C07284=1039.411,-98.894,424.242,168.623,36.335,156.842
C07285=1039.404,-99.143,424.252,168.620,36.336,156.842
C07286=1039.399,-99.393,424.262,168.618,36.336,156.842
C07287=1039.392,-99.680,424.273,168.615,36.336,156.842
C07288=1039.384,-99.967,424.285,168.612,36.337,156.842
C07289=1039.378,-100.255,424.297,168.609,36.337,156.842
C07290=1039.371,-100.541,424.308,168.606,36.338,156.842
C07291=1039.364,-100.791,424.319,168.603,36.338,156.842
C07292=1039.358,-101.041,424.329,168.601,36.338,156.842
C07293=1039.352,-101.291,424.338,168.598,36.338,156.842
C07294=1039.346,-101.540,424.349,168.596,36.339,156.842
C07295=1039.340,-101.790,424.359,168.593,36.340,156.843
C07296=1039.334,-102.040,424.368,168.591,36.340,156.843
C07297=1039.328,-102.289,424.379,168.589,36.340,156.843
C07298=1039.322,-102.539,424.389,168.586,36.340,156.843
C07299=1039.316,-102.789,424.398,168.584,36.341,156.843
C07300=1039.310,-103.038,424.409,168.581,36.341,156.843
C07301=1039.303,-103.288,424.418,168.579,36.342,156.843
C07302=1039.298,-103.538,424.428,168.576,36.341,156.843
C07303=1039.291,-103.787,424.439,168.574,36.342,156.843
C07304=1039.285,-104.037,424.448,168.571,36.343,156.843
C07305=1039.279,-104.287,424.458,168.568,36.343,156.843
C07306=1039.274,-104.537,424.468,168.566,36.343,156.843
C07307=1039.267,-104.786,424.478,168.563,36.343,156.843
C07308=1039.261,-105.036,424.488,168.561,36.344,156.843
C07309=1039.255,-105.286,424.497,168.558,36.345,156.844
C07310=1039.249,-105.536,424.508,168.556,36.345,156.844
C07311=1039.243,-105.786,424.517,168.553,36.345,156.844
C07312=1039.237,-106.035,424.528,168.550,36.345,156.844
C07313=1039.231,-106.285,424.537,168.548,36.346,156.844
C07314=1039.224,-106.535,424.547,168.545,36.347,156.844
C07315=1039.219,-106.785,424.557,168.543,36.347,156.844
C07316=1039.213,-107.034,424.566,168.540,36.347,156.844
C07317=1039.207,-107.284,424.576,168.538,36.348,156.844
C07318=1039.200,-107.533,424.586,168.535,36.348,156.844
C07319=1039.194,-107.783,424.596,168.532,36.349,156.844
C07320=1039.188,-108.033,424.605,168.530,36.349,156.844
C07321=1039.182,-108.283,424.616,168.528,36.350,156.844
C07322=1039.176,-108.533,424.625,168.526,36.350,156.844
C07323=1039.170,-108.783,424.635,168.523,36.350,156.845
C07324=1039.164,-109.033,424.644,168.520,36.351,156.845
C07325=1039.158,-109.282,424.654,168.518,36.352,156.845
C07326=1039.152,-109.532,424.663,168.515,36.352,156.845
C07327=1039.146,-109.781,424.673,168.513,36.352,156.845
C07328=1039.140,-110.031,424.682,168.510,36.353,156.845
C07329=1039.134,-110.281,424.692,168.507,36.354,156.845
C07330=1039.127,-110.531,424.701,168.505,36.354,156.845
C07331=1039.121,-110.780,424.711,168.502,36.354,156.845
C07332=1039.115,-111.030,424.720,168.499,36.355,156.845
C07333=1039.109,-111.280,424.730,168.497,36.356,156.845
C07334=1039.103,-111.530,424.740,168.494,36.356,156.846
C07335=1039.097,-111.780,424.749,168.492,36.356,156.846
C07336=1039.090,-112.029,424.759,168.489,36.357,156.846
C07337=1039.086,-112.279,424.768,168.486,36.357,156.846
C07338=1039.079,-112.529,424.778,168.484,36.358,156.846
C07339=1039.073,-112.778,424.788,168.481,36.359,156.846
C07340=1039.067,-113.028,424.797,168.479,36.359,156.846
C07341=1039.061,-113.278,424.807,168.477,36.359,156.846
C07342=1039.055,-113.528,424.816,168.474,36.360,156.846
C07343=1039.049,-113.778,424.826,168.472,36.361,156.846
C07344=1039.043,-114.027,424.835,168.469,36.361,156.847
C07345=1039.037,-114.276,424.845,168.467,36.362,156.847
C07346=1039.031,-114.526,424.854,168.464,36.362,156.847
C07347=1039.025,-114.777,424.863,168.461,36.363,156.847
C07348=1039.019,-115.027,424.873,168.459,36.363,156.847
C07349=1039.012,-115.276,424.882,168.456,36.364,156.847
C07350=1039.007,-115.525,424.891,168.453,36.365,156.847
C07351=1038.999,-115.812,424.902,168.450,36.365,156.847
C07352=1038.993,-116.098,424.913,168.447,36.366,156.847
C07353=1038.985,-116.385,424.923,168.444,36.367,156.847
C07354=1038.979,-116.671,424.934,168.441,36.367,156.848
C07355=1038.972,-116.921,424.943,168.439,36.368,156.848
C07356=1038.967,-117.170,424.952,168.436,36.368,156.848
C07357=1038.961,-117.420,424.962,168.434,36.369,156.848
C07358=1038.954,-117.670,424.972,168.432,36.370,156.848
C07359=1038.949,-117.920,424.980,168.429,36.370,156.848
C07360=1038.942,-118.169,424.989,168.427,36.371,156.848
C07361=1038.936,-118.419,424.999,168.424,36.372,156.848
C07362=1038.930,-118.669,425.007,168.421,36.372,156.848
C07363=1038.924,-118.919,425.017,168.419,36.373,156.849
C07364=1038.918,-119.168,425.026,168.416,36.374,156.849
C07365=1038.912,-119.418,425.036,168.413,36.374,156.849
C07366=1038.906,-119.668,425.045,168.411,36.375,156.849
C07367=1038.900,-119.918,425.054,168.408,36.376,156.849
C07368=1038.894,-120.167,425.063,168.405,36.376,156.849
C07369=1038.888,-120.417,425.072,168.403,36.377,156.849
C07370=1038.882,-120.667,425.081,168.400,36.378,156.849
C07371=1038.876,-120.917,425.091,168.398,36.378,156.849
C07372=1038.870,-121.167,425.099,168.395,36.379,156.850
C07373=1038.864,-121.416,425.108,168.393,36.379,156.850
C07374=1038.858,-121.666,425.117,168.391,36.380,156.850
C07375=1038.852,-121.916,425.126,168.388,36.381,156.850
C07376=1038.846,-122.165,425.136,168.385,36.381,156.850
C07377=1038.840,-122.416,425.145,168.383,36.382,156.850
C07378=1038.834,-122.665,425.153,168.380,36.383,156.850
C07379=1038.828,-122.915,425.162,168.377,36.384,156.851
C07380=1038.822,-123.165,425.172,168.375,36.385,156.851
C07381=1038.816,-123.414,425.181,168.372,36.385,156.851
C07382=1038.810,-123.664,425.189,168.369,36.386,156.851
C07383=1038.803,-123.914,425.199,168.367,36.387,156.851
C07384=1038.798,-124.163,425.207,168.364,36.387,156.851
C07385=1038.792,-124.413,425.217,168.361,36.388,156.851
C07386=1038.785,-124.663,425.225,168.359,36.389,156.851
C07387=1038.780,-124.912,425.234,168.357,36.389,156.851
C07388=1038.774,-125.163,425.243,168.354,36.391,156.852
C07389=1038.767,-125.412,425.252,168.352,36.391,156.852
C07390=1038.762,-125.662,425.261,168.349,36.392,156.852
C07391=1038.756,-125.912,425.270,168.346,36.392,156.852
C07392=1038.750,-126.161,425.278,168.344,36.393,156.852
C07393=1038.744,-126.412,425.287,168.341,36.394,156.852
C07394=1038.738,-126.661,425.296,168.338,36.395,156.852
C07395=1038.732,-126.911,425.304,168.336,36.396,156.853
C07396=1038.725,-127.161,425.314,168.333,36.396,156.853
C07397=1038.720,-127.410,425.322,168.330,36.397,156.853
C07398=1038.714,-127.661,425.331,168.328,36.398,156.853
C07399=1038.708,-127.910,425.340,168.326,36.399,156.853
C07400=1038.703,-128.160,425.350,168.324,36.399,156.853
C07401=1038.698,-128.409,425.360,168.321,36.399,156.853
C07402=1038.695,-128.658,425.370,168.318,36.398,156.853
C07403=1038.692,-128.909,425.382,168.316,36.397,156.853
C07404=1038.690,-129.158,425.393,168.314,36.396,156.853
C07405=1038.689,-129.409,425.406,168.312,36.394,156.852
C07406=1038.689,-129.658,425.419,168.311,36.391,156.852
C07407=1038.690,-129.909,425.433,168.308,36.388,156.851
C07408=1038.690,-130.159,425.447,168.307,36.384,156.851
C07409=1038.692,-130.409,425.462,168.306,36.381,156.850
C07410=1038.695,-130.659,425.477,168.304,36.377,156.849
C07411=1038.698,-130.909,425.493,168.303,36.372,156.849
C07412=1038.703,-131.160,425.510,168.301,36.367,156.848
C07413=1038.707,-131.409,425.527,168.301,36.361,156.847
C07414=1038.713,-131.660,425.545,168.300,36.355,156.846
C07415=1038.372,-131.683,425.279,168.252,36.557,156.880
C07416=1038.366,-131.435,425.261,168.253,36.564,156.881
C07417=1038.360,-131.184,425.244,168.254,36.569,156.882
C07418=1038.356,-130.934,425.227,168.255,36.574,156.883
C07419=1038.353,-130.683,425.212,168.256,36.579,156.883
C07420=1038.350,-130.434,425.195,168.258,36.584,156.884
C07421=1038.348,-130.184,425.181,168.259,36.587,156.885
C07422=1038.347,-129.933,425.166,168.261,36.591,156.885
C07423=1038.346,-129.683,425.153,168.263,36.593,156.886
C07424=1038.347,-129.433,425.140,168.264,36.596,156.886
C07425=1038.349,-129.184,425.127,168.266,36.598,156.887
C07426=1038.350,-128.934,425.115,168.269,36.600,156.887
C07427=1038.352,-128.683,425.104,168.271,36.601,156.887
C07428=1038.357,-128.434,425.093,168.273,36.601,156.887
C07429=1038.361,-128.184,425.083,168.276,36.602,156.887
C07430=1038.365,-127.934,425.074,168.278,36.601,156.887
C07431=1038.371,-127.685,425.065,168.281,36.601,156.887
C07432=1038.377,-127.435,425.056,168.283,36.600,156.887
C07433=1038.383,-127.185,425.047,168.286,36.599,156.887
C07434=1038.389,-126.935,425.038,168.288,36.598,156.887
C07435=1038.395,-126.686,425.030,168.291,36.597,156.887
C07436=1038.401,-126.436,425.021,168.293,36.597,156.886
C07437=1038.407,-126.185,425.012,168.296,36.596,156.886
C07438=1038.413,-125.937,425.003,168.299,36.595,156.886
C07439=1038.419,-125.686,424.995,168.301,36.594,156.886
C07440=1038.425,-125.437,424.985,168.304,36.593,156.886
C07441=1038.431,-125.187,424.977,168.307,36.593,156.886
C07442=1038.437,-124.937,424.968,168.309,36.592,156.886
C07443=1038.443,-124.688,424.959,168.312,36.591,156.885
C07444=1038.450,-124.438,424.950,168.315,36.590,156.885
C07445=1038.455,-124.188,424.941,168.317,36.589,156.885
C07446=1038.461,-123.939,424.932,168.320,36.589,156.885
C07447=1038.467,-123.688,424.923,168.322,36.588,156.885
C07448=1038.474,-123.439,424.914,168.324,36.587,156.885
C07449=1038.479,-123.189,424.906,168.327,36.587,156.885
C07450=1038.485,-122.939,424.896,168.330,36.585,156.885
C07451=1038.491,-122.689,424.887,168.332,36.585,156.884
C07452=1038.497,-122.440,424.878,168.335,36.584,156.884
C07453=1038.504,-122.190,424.869,168.338,36.583,156.884
C07454=1038.509,-121.940,424.860,168.340,36.583,156.884
C07455=1038.515,-121.691,424.851,168.343,36.582,156.884
C07456=1038.521,-121.440,424.842,168.346,36.581,156.884
C07457=1038.527,-121.190,424.833,168.348,36.581,156.884
C07458=1038.533,-120.942,424.824,168.351,36.580,156.884
C07459=1038.539,-120.691,424.815,168.354,36.579,156.884
C07460=1038.545,-120.441,424.806,168.355,36.578,156.883
C07461=1038.551,-120.192,424.796,168.358,36.577,156.883
C07462=1038.557,-119.942,424.788,168.361,36.577,156.883
C07463=1038.563,-119.692,424.778,168.363,36.576,156.883
C07464=1038.570,-119.443,424.769,168.366,36.575,156.883
C07465=1038.575,-119.193,424.761,168.369,36.575,156.883
C07466=1038.581,-118.943,424.751,168.371,36.574,156.883
C07467=1038.587,-118.693,424.741,168.374,36.573,156.883
C07468=1038.593,-118.443,424.733,168.377,36.573,156.882
C07469=1038.599,-118.194,424.723,168.379,36.572,156.882
C07470=1038.605,-117.944,424.714,168.382,36.571,156.882
C07471=1038.612,-117.694,424.705,168.385,36.571,156.882
C07472=1038.618,-117.444,424.696,168.387,36.570,156.882
C07473=1038.623,-117.195,424.687,168.390,36.569,156.882
C07474=1038.630,-116.945,424.677,168.392,36.569,156.882
C07475=1038.636,-116.695,424.668,168.394,36.568,156.882
C07476=1038.642,-116.409,424.657,168.397,36.567,156.882
C07477=1038.650,-116.122,424.646,168.400,36.567,156.881
C07478=1038.657,-115.836,424.636,168.403,36.566,156.881
C07479=1038.663,-115.550,424.625,168.406,36.565,156.881
C07480=1038.670,-115.300,424.616,168.409,36.565,156.881
C07481=1038.676,-115.051,424.607,168.412,36.564,156.881
C07482=1038.682,-114.801,424.597,168.414,36.563,156.881
C07483=1038.688,-114.550,424.588,168.417,36.563,156.881
C07484=1038.694,-114.301,424.579,168.420,36.562,156.881
C07485=1038.700,-114.052,424.569,168.422,36.562,156.881
C07486=1038.706,-113.802,424.560,168.425,36.561,156.880
C07487=1038.712,-113.552,424.550,168.427,36.560,156.880
C07488=1038.718,-113.302,424.541,168.430,36.560,156.880
C07489=1038.724,-113.052,424.531,168.433,36.560,156.880
C07490=1038.730,-112.803,424.522,168.434,36.559,156.880
C07491=1038.736,-112.553,424.512,168.437,36.558,156.880
C07492=1038.742,-112.304,424.503,168.440,36.558,156.880
C07493=1038.748,-112.054,424.493,168.442,36.557,156.880
C07494=1038.753,-111.803,424.484,168.445,36.556,156.880
C07495=1038.760,-111.553,424.474,168.447,36.556,156.880
C07496=1038.766,-111.304,424.465,168.450,36.556,156.880
C07497=1038.772,-111.054,424.455,168.453,36.555,156.880
C07498=1038.778,-110.804,424.446,168.455,36.554,156.879
C07499=1038.784,-110.555,424.436,168.458,36.554,156.879
C07500=1038.790,-110.305,424.427,168.461,36.553,156.879
C07501=1038.796,-110.055,424.417,168.463,36.553,156.879
C07502=1038.802,-109.805,424.408,168.466,36.552,156.879
C07503=1038.809,-109.556,424.397,168.468,36.552,156.879
C07504=1038.815,-109.306,424.388,168.471,36.551,156.879
C07505=1038.821,-109.057,424.378,168.474,36.550,156.879
C07506=1038.827,-108.807,424.369,168.476,36.550,156.879
C07507=1038.833,-108.557,424.359,168.479,36.550,156.879
C07508=1038.840,-108.307,424.349,168.481,36.549,156.879
C07509=1038.845,-108.057,424.339,168.483,36.548,156.878
C07510=1038.851,-107.807,424.330,168.486,36.548,156.878
C07511=1038.857,-107.558,424.320,168.488,36.548,156.878
C07512=1038.864,-107.308,424.311,168.491,36.547,156.878
C07513=1038.870,-107.058,424.301,168.494,36.546,156.878
C07514=1038.876,-106.810,424.291,168.496,36.546,156.878
C07515=1038.882,-106.560,424.282,168.499,36.546,156.878
C07516=1038.887,-106.310,424.271,168.501,36.545,156.878
C07517=1038.893,-106.060,424.262,168.504,36.544,156.878
C07518=1038.900,-105.810,424.252,168.507,36.544,156.878
C07519=1038.906,-105.560,424.243,168.509,36.544,156.878
C07520=1038.911,-105.311,424.232,168.512,36.543,156.878
C07521=1038.918,-105.061,424.222,168.514,36.543,156.878
C07522=1038.924,-104.811,424.213,168.517,36.542,156.877
C07523=1038.930,-104.561,424.203,168.520,36.542,156.877
C07524=1038.936,-104.312,424.192,168.522,36.542,156.877
C07525=1038.942,-104.062,424.183,168.525,36.541,156.877
C07526=1038.948,-103.812,424.173,168.527,36.541,156.877
C07527=1038.954,-103.562,424.164,168.530,36.540,156.877
C07528=1038.960,-103.313,424.153,168.532,36.540,156.877
C07529=1038.966,-103.063,424.143,168.535,36.540,156.877
C07530=1038.972,-102.813,424.134,168.537,36.539,156.877
C07531=1038.979,-102.564,424.123,168.539,36.539,156.877
C07532=1038.985,-102.313,424.113,168.542,36.538,156.877
C07533=1038.991,-102.064,424.103,168.544,36.538,156.877
C07534=1038.997,-101.814,424.094,168.547,36.538,156.877
C07535=1039.003,-101.564,424.083,168.550,36.537,156.877
C07536=1039.009,-101.314,424.073,168.552,36.537,156.877
C07537=1039.016,-101.065,424.063,168.555,36.536,156.876
C07538=1039.022,-100.816,424.053,168.557,36.536,156.876
C07539=1039.027,-100.565,424.043,168.560,36.536,156.876
C07540=1039.035,-100.279,424.031,168.563,36.535,156.876
C07541=1039.042,-99.991,424.020,168.566,36.534,156.876
C07542=1039.049,-99.704,424.008,168.569,36.534,156.876
C07543=1039.055,-99.417,423.997,168.572,36.534,156.876
C07544=1039.062,-99.167,423.987,168.574,36.534,156.876
C07545=1039.068,-98.917,423.976,168.577,36.533,156.876
C07546=1039.074,-98.668,423.966,168.579,36.532,156.876
C07547=1039.081,-98.418,423.957,168.582,36.532,156.876
C07548=1039.086,-98.168,423.946,168.585,36.532,156.876
C07549=1039.092,-97.919,423.936,168.587,36.532,156.876
C07550=1039.099,-97.669,423.927,168.590,36.531,156.875
C07551=1039.105,-97.419,423.915,168.592,36.531,156.875
C07552=1039.111,-97.169,423.906,168.595,36.531,156.875
C07553=1039.117,-96.920,423.895,168.597,36.531,156.875
C07554=1039.123,-96.670,423.885,168.600,36.531,156.875
C07555=1039.129,-96.420,423.874,168.602,36.530,156.875
C07556=1039.135,-96.171,423.864,168.605,36.530,156.875
C07557=1039.141,-95.921,423.854,168.607,36.530,156.875
C07558=1039.146,-95.672,423.843,168.609,36.529,156.875
C07559=1039.153,-95.421,423.833,168.611,36.529,156.875
C07560=1039.159,-95.172,423.822,168.614,36.529,156.875
C07561=1039.165,-94.922,423.812,168.617,36.529,156.875
C07562=1039.171,-94.672,423.802,168.619,36.529,156.875
C07563=1039.177,-94.423,423.791,168.622,36.529,156.875
C07564=1039.183,-94.174,423.781,168.624,36.528,156.875
C07565=1039.189,-93.923,423.770,168.627,36.528,156.875
C07566=1039.196,-93.674,423.760,168.629,36.528,156.875
C07567=1039.201,-93.423,423.750,168.632,36.527,156.875
C07568=1039.207,-93.174,423.739,168.634,36.527,156.875
C07569=1039.213,-92.925,423.729,168.637,36.527,156.875
C07570=1039.219,-92.675,423.718,168.639,36.527,156.875
C07571=1039.226,-92.425,423.708,168.642,36.527,156.875
C07572=1039.231,-92.175,423.697,168.644,36.527,156.875
C07573=1039.238,-91.926,423.687,168.647,36.526,156.875
C07574=1039.243,-91.676,423.676,168.649,36.526,156.875
C07575=1039.250,-91.426,423.665,168.652,36.526,156.875
C07576=1039.256,-91.177,423.655,168.654,36.525,156.874
C07577=1039.262,-90.927,423.644,168.657,36.525,156.874
C07578=1039.268,-90.677,423.634,168.659,36.525,156.874
C07579=1039.274,-90.427,423.623,168.662,36.525,156.874
C07580=1039.280,-90.178,423.612,168.664,36.525,156.874
C07581=1039.287,-89.929,423.602,168.667,36.525,156.874
C07582=1039.292,-89.678,423.592,168.669,36.525,156.874
C07583=1039.299,-89.429,423.581,168.672,36.524,156.874
C07584=1039.305,-89.179,423.570,168.674,36.524,156.874
C07585=1039.311,-88.930,423.560,168.677,36.524,156.874
C07586=1039.318,-88.680,423.549,168.680,36.523,156.874
C07587=1039.323,-88.430,423.539,168.682,36.523,156.874
C07588=1039.329,-88.180,423.528,168.685,36.523,156.874
C07589=1039.335,-87.931,423.518,168.687,36.523,156.874
C07590=1039.342,-87.681,423.506,168.690,36.523,156.874
C07591=1039.348,-87.432,423.496,168.692,36.523,156.874
C07592=1039.354,-87.182,423.485,168.695,36.523,156.874
C07593=1039.360,-86.932,423.474,168.697,36.523,156.874
C07594=1039.366,-86.682,423.464,168.700,36.522,156.874
C07595=1039.372,-86.433,423.453,168.702,36.522,156.874
C07596=1039.379,-86.182,423.442,168.705,36.522,156.874
C07597=1039.385,-85.933,423.432,168.707,36.522,156.874
C07598=1039.391,-85.683,423.421,168.710,36.521,156.874
C07599=1039.397,-85.434,423.410,168.712,36.521,156.874
C07600=1039.404,-85.184,423.400,168.715,36.521,156.874
C07601=1039.410,-84.934,423.388,168.717,36.521,156.874
C07602=1039.416,-84.685,423.377,168.720,36.521,156.874
C07603=1039.422,-84.436,423.367,168.722,36.521,156.874
C07604=1039.429,-84.150,423.355,168.725,36.521,156.874
C07605=1039.437,-83.865,423.343,168.728,36.521,156.874
C07606=1039.444,-83.580,423.331,168.731,36.520,156.874
C07607=1039.450,-83.295,423.317,168.733,36.520,156.874
C07608=1039.457,-83.046,423.307,168.736,36.520,156.874
C07609=1039.463,-82.796,423.295,168.738,36.520,156.874
C07610=1039.469,-82.546,423.285,168.741,36.520,156.874
C07611=1039.476,-82.296,423.274,168.742,36.519,156.873
C07612=1039.482,-82.047,423.263,168.745,36.519,156.873
C07613=1039.488,-81.797,423.252,168.747,36.519,156.873
C07614=1039.495,-81.548,423.242,168.750,36.519,156.873
C07615=1039.501,-81.297,423.230,168.752,36.519,156.873
C07616=1039.507,-81.048,423.219,168.755,36.519,156.873
C07617=1039.513,-80.799,423.209,168.757,36.519,156.873
C07618=1039.519,-80.548,423.198,168.760,36.519,156.873
C07619=1039.525,-80.299,423.187,168.762,36.519,156.873
C07620=1039.532,-80.049,423.176,168.765,36.519,156.873
C07621=1039.538,-79.800,423.165,168.767,36.518,156.873
C07622=1039.545,-79.550,423.153,168.770,36.518,156.873
C07623=1039.550,-79.301,423.143,168.772,36.518,156.873
C07624=1039.557,-79.050,423.131,168.775,36.518,156.873
C07625=1039.563,-78.801,423.120,168.777,36.518,156.873
C07626=1039.569,-78.551,423.109,168.780,36.518,156.873
C07627=1039.575,-78.302,423.098,168.782,36.518,156.873
C07628=1039.581,-78.052,423.086,168.784,36.518,156.873
C07629=1039.587,-77.802,423.076,168.787,36.518,156.873
C07630=1039.593,-77.552,423.064,168.789,36.518,156.873
C07631=1039.600,-77.303,423.053,168.792,36.518,156.873
C07632=1039.606,-77.053,423.042,168.794,36.518,156.873
C07633=1039.612,-76.804,423.031,168.797,36.518,156.873
C07634=1039.619,-76.553,423.020,168.799,36.518,156.873
C07635=1039.625,-76.305,423.008,168.802,36.518,156.873
C07636=1039.631,-76.054,422.997,168.804,36.518,156.873
C07637=1039.637,-75.805,422.986,168.806,36.518,156.873
C07638=1039.643,-75.555,422.974,168.809,36.518,156.873
C07639=1039.649,-75.306,422.963,168.811,36.518,156.873
C07640=1039.655,-75.056,422.952,168.814,36.519,156.873
C07641=1039.662,-74.806,422.940,168.816,36.519,156.873
C07642=1039.668,-74.557,422.929,168.819,36.519,156.873
C07643=1039.674,-74.306,422.918,168.821,36.519,156.873
C07644=1039.680,-74.058,422.906,168.823,36.519,156.873
C07645=1039.686,-73.807,422.895,168.826,36.519,156.873
C07646=1039.692,-73.558,422.884,168.828,36.519,156.873
C07647=1039.699,-73.308,422.872,168.831,36.519,156.873
C07648=1039.704,-73.058,422.861,168.833,36.519,156.873
C07649=1039.711,-72.809,422.849,168.835,36.519,156.873
C07650=1039.717,-72.559,422.838,168.838,36.519,156.873
C07651=1039.723,-72.310,422.826,168.840,36.519,156.873
C07652=1039.729,-72.059,422.814,168.843,36.519,156.873
C07653=1039.735,-71.811,422.803,168.846,36.520,156.874
C07654=1039.741,-71.560,422.791,168.848,36.520,156.874
C07655=1039.747,-71.311,422.780,168.851,36.520,156.874
C07656=1039.753,-71.061,422.769,168.853,36.520,156.874
C07657=1039.759,-70.811,422.756,168.856,36.520,156.874
C07658=1039.765,-70.562,422.745,168.858,36.521,156.874
C07659=1039.772,-70.312,422.733,168.860,36.521,156.874
C07660=1039.777,-70.063,422.722,168.863,36.521,156.874
C07661=1039.783,-69.813,422.710,168.865,36.521,156.874
C07662=1039.790,-69.563,422.699,168.867,36.521,156.874
C07663=1039.796,-69.314,422.687,168.870,36.521,156.874
C07664=1039.802,-69.064,422.676,168.872,36.521,156.874
C07665=1039.807,-68.814,422.664,168.875,36.521,156.874
C07666=1039.814,-68.565,422.652,168.877,36.522,156.874
C07667=1039.820,-68.315,422.640,168.879,36.522,156.874
C07668=1039.827,-68.032,422.627,168.882,36.522,156.874
C07669=1039.834,-67.750,422.614,168.885,36.523,156.874
C07670=1039.841,-67.467,422.600,168.887,36.523,156.874
C07671=1039.848,-67.184,422.587,168.890,36.523,156.874
C07672=1039.855,-66.934,422.575,168.892,36.523,156.874
C07673=1039.860,-66.685,422.564,168.895,36.523,156.874
C07674=1039.866,-66.435,422.552,168.897,36.523,156.874
C07675=1039.873,-66.185,422.540,168.900,36.523,156.874
C07676=1039.878,-65.936,422.528,168.902,36.523,156.874
C07677=1039.885,-65.686,422.516,168.904,36.524,156.874
C07678=1039.891,-65.436,422.505,168.907,36.524,156.874
C07679=1039.897,-65.187,422.494,168.909,36.524,156.874
C07680=1039.903,-64.937,422.481,168.911,36.524,156.874
C07681=1039.910,-64.688,422.469,168.914,36.524,156.874
C07682=1039.916,-64.437,422.458,168.916,36.524,156.874
C07683=1039.921,-64.188,422.446,168.918,36.524,156.874
C07684=1039.928,-63.939,422.434,168.921,36.525,156.875
C07685=1039.935,-63.689,422.422,168.923,36.525,156.875
C07686=1039.941,-63.439,422.411,168.925,36.525,156.875
C07687=1039.946,-63.190,422.398,168.928,36.526,156.875
C07688=1039.953,-62.940,422.386,168.930,36.526,156.875
C07689=1039.960,-62.691,422.374,168.933,36.526,156.875
C07690=1039.965,-62.441,422.362,168.935,36.526,156.875
C07691=1039.971,-62.191,422.351,168.937,36.526,156.875
C07692=1039.978,-61.942,422.339,168.940,36.526,156.875
C07693=1039.984,-61.692,422.327,168.942,36.526,156.875
C07694=1039.990,-61.442,422.315,168.944,36.527,156.875
C07695=1039.997,-61.193,422.303,168.947,36.527,156.875
C07696=1040.003,-60.944,422.291,168.949,36.527,156.875
C07697=1040.009,-60.693,422.279,168.951,36.528,156.875
C07698=1040.015,-60.444,422.267,168.954,36.528,156.875
C07699=1040.022,-60.194,422.255,168.956,36.528,156.875
C07700=1040.028,-59.944,422.243,168.958,36.528,156.875
C07701=1040.035,-59.695,422.231,168.961,36.528,156.875
C07702=1040.041,-59.446,422.219,168.963,36.528,156.875
C07703=1040.046,-59.196,422.207,168.966,36.529,156.875
C07704=1040.053,-58.946,422.195,168.969,36.529,156.875
C07705=1040.059,-58.696,422.183,168.971,36.529,156.875
C07706=1040.065,-58.446,422.171,168.973,36.530,156.875
C07707=1040.072,-58.197,422.159,168.976,36.530,156.875
C07708=1040.079,-57.947,422.147,168.978,36.530,156.875
C07709=1040.084,-57.698,422.135,168.980,36.530,156.875
C07710=1040.091,-57.448,422.123,168.983,36.530,156.875
C07711=1040.097,-57.199,422.111,168.985,36.530,156.875
C07712=1040.103,-56.949,422.098,168.987,36.531,156.876
C07713=1040.110,-56.699,422.086,168.990,36.531,156.876
C07714=1040.116,-56.450,422.074,168.992,36.531,156.876
C07715=1040.122,-56.200,422.062,168.994,36.532,156.876
C07716=1040.129,-55.935,422.049,168.997,36.532,156.876
C07717=1040.136,-55.671,422.037,168.999,36.532,156.876
C07718=1040.143,-55.405,422.023,169.002,36.532,156.876
C07719=1040.150,-55.141,422.010,169.004,36.532,156.876
C07720=1040.156,-54.891,421.998,169.007,36.533,156.876
C07721=1040.162,-54.641,421.985,169.009,36.533,156.876
C07722=1040.169,-54.392,421.973,169.011,36.533,156.876
C07723=1040.175,-54.142,421.961,169.014,36.533,156.876
C07724=1040.181,-53.892,421.949,169.016,36.533,156.876
C07725=1040.188,-53.643,421.937,169.018,36.533,156.876
C07726=1040.194,-53.393,421.924,169.021,36.534,156.876
C07727=1040.201,-53.143,421.912,169.023,36.534,156.876
C07728=1040.207,-52.894,421.901,169.025,36.535,156.876
C07729=1040.213,-52.644,421.888,169.028,36.535,156.876
C07730=1040.220,-52.394,421.876,169.030,36.535,156.876
C07731=1040.226,-52.145,421.863,169.032,36.535,156.876
C07732=1040.233,-51.879,421.851,169.035,36.535,156.876
C07733=1040.239,-51.613,421.838,169.037,36.536,156.876
C07734=1040.247,-51.346,421.824,169.040,36.536,156.876
C07735=1040.253,-51.080,421.811,169.042,36.536,156.876
C07736=1040.260,-50.831,421.799,169.044,36.537,156.877
C07737=1040.266,-50.581,421.786,169.047,36.537,156.877
C07738=1040.272,-50.332,421.774,169.049,36.537,156.877
C07739=1040.278,-50.082,421.761,169.051,36.537,156.877
C07740=1040.284,-49.832,421.749,169.053,36.538,156.877
C07741=1040.291,-49.583,421.736,169.057,36.539,156.877
C07742=1040.297,-49.333,421.724,169.059,36.539,156.877
C07743=1040.303,-49.083,421.711,169.061,36.539,156.877
C07744=1040.309,-48.834,421.698,169.063,36.539,156.877
C07745=1040.316,-48.584,421.686,169.066,36.540,156.877
C07746=1040.322,-48.335,421.673,169.068,36.541,156.877
C07747=1040.328,-48.085,421.660,169.070,36.541,156.877
C07748=1040.334,-47.835,421.647,169.072,36.541,156.877
C07749=1040.341,-47.586,421.636,169.075,36.542,156.878
C07750=1040.347,-47.337,421.622,169.077,36.542,156.878
C07751=1040.353,-47.087,421.610,169.079,36.542,156.878
C07752=1040.359,-46.837,421.597,169.081,36.542,156.878
C07753=1040.366,-46.588,421.584,169.084,36.543,156.878
C07754=1040.372,-46.337,421.572,169.086,36.544,156.878
C07755=1040.378,-46.087,421.559,169.088,36.544,156.878
C07756=1040.384,-45.838,421.546,169.090,36.544,156.878
C07757=1040.391,-45.589,421.534,169.093,36.545,156.878
C07758=1040.397,-45.339,421.520,169.095,36.545,156.878
C07759=1040.403,-45.089,421.508,169.097,36.546,156.878
C07760=1040.409,-44.840,421.495,169.099,36.546,156.878
C07761=1040.416,-44.591,421.483,169.102,36.546,156.878
C07762=1040.422,-44.341,421.470,169.104,36.547,156.878
C07763=1040.428,-44.091,421.457,169.106,36.547,156.878
C07764=1040.434,-43.842,421.444,169.109,36.548,156.879
C07765=1040.441,-43.593,421.432,169.112,36.548,156.879
C07766=1040.447,-43.342,421.419,169.114,36.548,156.879
C07767=1040.454,-43.093,421.405,169.116,36.549,156.879
C07768=1040.459,-42.843,421.393,169.118,36.550,156.879
C07769=1040.466,-42.594,421.380,169.120,36.550,156.879
C07770=1040.472,-42.344,421.368,169.123,36.550,156.879
C07771=1040.479,-42.095,421.354,169.125,36.551,156.879
C07772=1040.484,-41.845,421.342,169.127,36.551,156.879
C07773=1040.491,-41.596,421.329,169.129,36.551,156.879
C07774=1040.497,-41.346,421.315,169.132,36.552,156.879
C07775=1040.504,-41.096,421.303,169.134,36.552,156.879
C07776=1040.510,-40.847,421.290,169.136,36.553,156.879
C07777=1040.516,-40.597,421.277,169.138,36.553,156.880
C07778=1040.522,-40.348,421.264,169.140,36.553,156.880
C07779=1040.529,-40.097,421.251,169.143,36.554,156.880
C07780=1040.536,-39.848,421.238,169.145,36.555,156.880
C07781=1040.542,-39.599,421.225,169.147,36.555,156.880
C07782=1040.548,-39.349,421.212,169.149,36.555,156.880
C07783=1040.554,-39.100,421.199,169.152,36.556,156.880
C07784=1040.561,-38.850,421.186,169.154,36.556,156.880
C07785=1040.567,-38.600,421.173,169.157,36.557,156.880
C07786=1040.573,-38.351,421.160,169.159,36.557,156.880
C07787=1040.579,-38.101,421.146,169.161,36.558,156.880
C07788=1040.585,-37.851,421.134,169.163,36.558,156.881
C07789=1040.592,-37.602,421.121,169.166,36.558,156.881
C07790=1040.598,-37.352,421.107,169.168,36.559,156.881
C07791=1040.604,-37.102,421.094,169.170,36.560,156.881
C07792=1040.610,-36.853,421.081,169.172,36.560,156.881
C07793=1040.617,-36.604,421.068,169.174,36.561,156.881
C07794=1040.623,-36.355,421.055,169.177,36.562,156.881
C07795=1040.629,-36.104,421.042,169.179,36.562,156.881
C07796=1040.636,-35.824,421.027,169.181,36.562,156.881
C07797=1040.643,-35.542,421.012,169.184,36.563,156.881
C07798=1040.651,-35.261,420.997,169.186,36.564,156.881
C07799=1040.657,-34.980,420.982,169.188,36.564,156.882
C07800=1040.664,-34.730,420.968,169.191,36.565,156.882
C07801=1040.670,-34.481,420.955,169.193,36.566,156.882
C07802=1040.676,-34.232,420.942,169.196,36.566,156.882
C07803=1040.683,-33.982,420.928,169.198,36.567,156.882
C07804=1040.689,-33.732,420.916,169.200,36.567,156.882
C07805=1040.695,-33.483,420.902,169.202,36.567,156.882
C07806=1040.701,-33.233,420.889,169.205,36.568,156.882
C07807=1040.708,-32.983,420.876,169.207,36.569,156.882
C07808=1040.714,-32.734,420.862,169.209,36.569,156.883
C07809=1040.720,-32.485,420.849,169.211,36.570,156.883
C07810=1040.727,-32.235,420.835,169.213,36.571,156.883
C07811=1040.733,-31.986,420.822,169.215,36.571,156.883
C07812=1040.740,-31.736,420.809,169.218,36.571,156.883
C07813=1040.745,-31.486,420.796,169.220,36.572,156.883
C07814=1040.752,-31.236,420.782,169.222,36.573,156.883
C07815=1040.758,-30.987,420.769,169.224,36.573,156.883
C07816=1040.764,-30.738,420.756,169.226,36.574,156.883
C07817=1040.771,-30.488,420.742,169.228,36.574,156.883
C07818=1040.777,-30.239,420.729,169.230,36.574,156.883
C07819=1040.783,-29.989,420.715,169.234,36.575,156.884
C07820=1040.790,-29.739,420.702,169.236,36.576,156.884
C07821=1040.796,-29.490,420.688,169.238,36.576,156.884
C07822=1040.803,-29.240,420.675,169.240,36.577,156.884
C07823=1040.809,-28.991,420.662,169.242,36.578,156.884
C07824=1040.815,-28.741,420.648,169.244,36.578,156.884
C07825=1040.822,-28.491,420.634,169.246,36.578,156.884
C07826=1040.828,-28.242,420.621,169.249,36.579,156.884
C07827=1040.834,-27.993,420.608,169.251,36.580,156.884
C07828=1040.841,-27.743,420.594,169.253,36.580,156.884
C07829=1040.847,-27.494,420.581,169.255,36.581,156.885
C07830=1040.854,-27.244,420.567,169.257,36.581,156.885
C07831=1040.860,-26.994,420.554,169.259,36.582,156.885
C07832=1040.866,-26.745,420.540,169.261,36.583,156.885
C07833=1040.873,-26.495,420.526,169.263,36.583,156.885
C07834=1040.879,-26.246,420.512,169.267,36.584,156.885
C07835=1040.884,-25.997,420.498,169.269,36.585,156.885
C07836=1040.891,-25.747,420.485,169.271,36.585,156.885
C07837=1040.897,-25.497,420.471,169.273,36.586,156.886
C07838=1040.904,-25.247,420.457,169.275,36.587,156.886
C07839=1040.910,-24.998,420.444,169.277,36.587,156.886
C07840=1040.916,-24.749,420.429,169.279,36.588,156.886
C07841=1040.922,-24.499,420.416,169.281,36.589,156.886
C07842=1040.929,-24.250,420.402,169.283,36.589,156.886
C07843=1040.935,-23.999,420.388,169.285,36.590,156.886
C07844=1040.941,-23.750,420.375,169.288,36.590,156.886
C07845=1040.947,-23.501,420.361,169.290,36.591,156.886
C07846=1040.953,-23.251,420.347,169.292,36.592,156.887
C07847=1040.960,-23.002,420.333,169.294,36.592,156.887
C07848=1040.966,-22.752,420.320,169.297,36.593,156.887
C07849=1040.972,-22.503,420.305,169.299,36.594,156.887
C07850=1040.979,-22.253,420.292,169.301,36.594,156.887
C07851=1040.985,-22.003,420.278,169.303,36.595,156.887
C07852=1040.991,-21.753,420.264,169.305,36.596,156.887
C07853=1040.998,-21.505,420.250,169.307,36.596,156.887
C07854=1041.004,-21.255,420.236,169.309,36.597,156.888
C07855=1041.010,-21.005,420.223,169.311,36.597,156.888
C07856=1041.017,-20.756,420.208,169.314,36.598,156.888
C07857=1041.023,-20.506,420.194,169.316,36.599,156.888
C07858=1041.030,-20.256,420.181,169.318,36.599,156.888
C07859=1041.035,-20.007,420.167,169.320,36.600,156.888
C07860=1041.043,-19.725,420.151,169.322,36.601,156.888
C07861=1041.050,-19.444,420.135,169.324,36.601,156.888
C07862=1041.057,-19.161,420.120,169.328,36.603,156.889
C07863=1041.064,-18.880,420.104,169.330,36.603,156.889
C07864=1041.070,-18.630,420.090,169.332,36.604,156.889
C07865=1041.077,-18.381,420.075,169.334,36.604,156.889
C07866=1041.083,-18.131,420.062,169.336,36.605,156.889
C07867=1041.089,-17.881,420.048,169.338,36.606,156.889
C07868=1041.096,-17.632,420.034,169.340,36.606,156.889
C07869=1041.102,-17.383,420.020,169.343,36.607,156.889
C07870=1041.109,-17.133,420.005,169.345,36.608,156.890
C07871=1041.115,-16.884,419.992,169.347,36.608,156.890
C07872=1041.121,-16.634,419.977,169.349,36.609,156.890
C07873=1041.128,-16.385,419.964,169.351,36.610,156.890
C07874=1041.134,-16.135,419.950,169.353,36.610,156.890
C07875=1041.140,-15.886,419.936,169.356,36.611,156.890
C07876=1041.147,-15.636,419.922,169.358,36.611,156.890
C07877=1041.153,-15.386,419.907,169.360,36.612,156.890
C07878=1041.160,-15.137,419.894,169.362,36.613,156.890
C07879=1041.166,-14.887,419.879,169.364,36.614,156.891
C07880=1041.172,-14.638,419.865,169.366,36.615,156.891
C07881=1041.179,-14.388,419.851,169.368,36.615,156.891
C07882=1041.184,-14.139,419.837,169.370,36.616,156.891
C07883=1041.191,-13.889,419.822,169.372,36.617,156.891
C07884=1041.198,-13.640,419.807,169.374,36.617,156.891
C07885=1041.203,-13.390,419.794,169.376,36.618,156.891
C07886=1041.210,-13.140,419.779,169.378,36.619,156.892
C07887=1041.216,-12.891,419.765,169.381,36.620,156.892
C07888=1041.222,-12.642,419.750,169.383,36.620,156.892
C07889=1041.228,-12.392,419.735,169.385,36.621,156.892
C07890=1041.235,-12.143,419.722,169.387,36.622,156.892
C07891=1041.241,-11.893,419.707,169.389,36.623,156.892
C07892=1041.247,-11.643,419.693,169.391,36.623,156.892
C07893=1041.254,-11.394,419.679,169.393,36.624,156.893
C07894=1041.260,-11.144,419.664,169.395,36.625,156.893
C07895=1041.266,-10.895,419.650,169.397,36.625,156.893
C07896=1041.273,-10.645,419.636,169.399,36.627,156.893
C07897=1041.279,-10.396,419.621,169.401,36.627,156.893
C07898=1041.285,-10.146,419.607,169.403,36.628,156.893
C07899=1041.292,-9.897,419.593,169.406,36.629,156.893
C07900=1041.298,-9.647,419.578,169.408,36.629,156.893
C07901=1041.304,-9.398,419.563,169.410,36.630,156.894
C07902=1041.311,-9.148,419.550,169.412,36.631,156.894
C07903=1041.317,-8.899,419.535,169.414,36.632,156.894
C07904=1041.323,-8.650,419.520,169.416,36.632,156.894
C07905=1041.330,-8.400,419.506,169.418,36.633,156.894
C07906=1041.336,-8.150,419.491,169.420,36.634,156.894
C07907=1041.342,-7.901,419.477,169.422,36.635,156.895
C07908=1041.348,-7.651,419.462,169.424,36.636,156.895
C07909=1041.355,-7.402,419.448,169.426,36.636,156.895
C07910=1041.361,-7.153,419.434,169.428,36.637,156.895
C07911=1041.367,-6.903,419.419,169.431,36.637,156.895
C07912=1041.374,-6.654,419.404,169.433,36.639,156.895
C07913=1041.381,-6.404,419.389,169.435,36.639,156.895
C07914=1041.386,-6.154,419.376,169.437,36.640,156.895
C07915=1041.393,-5.905,419.361,169.439,36.641,156.896
C07916=1041.400,-5.655,419.346,169.441,36.641,156.896
C07917=1041.405,-5.406,419.332,169.443,36.642,156.896
C07918=1041.412,-5.157,419.317,169.445,36.643,156.896
C07919=1041.419,-4.907,419.302,169.447,36.644,156.896
C07920=1041.425,-4.657,419.288,169.449,36.644,156.896
C07921=1041.431,-4.407,419.273,169.451,36.645,156.896
C07922=1041.437,-4.158,419.259,169.453,36.646,156.897
C07923=1041.444,-3.909,419.244,169.456,36.647,156.897
C07924=1041.451,-3.626,419.228,169.459,36.648,156.897
C07925=1041.459,-3.343,419.211,169.461,36.648,156.897
C07926=1041.466,-3.058,419.194,169.463,36.649,156.897
C07927=1041.473,-2.775,419.177,169.465,36.651,156.897
C07928=1041.479,-2.526,419.163,169.467,36.651,156.898
C07929=1041.485,-2.276,419.148,169.469,36.652,156.898
C07930=1041.491,-2.027,419.133,169.471,36.653,156.898
C07931=1041.498,-1.777,419.118,169.473,36.654,156.898
C07932=1041.503,-1.528,419.103,169.476,36.655,156.898
C07933=1041.510,-1.278,419.088,169.478,36.656,156.898
C07934=1041.516,-1.029,419.073,169.480,36.656,156.899
C07935=1041.523,-0.779,419.058,169.482,36.658,156.899
C07936=1041.529,-0.531,419.043,169.484,36.658,156.899
C07937=1041.535,-0.281,419.028,169.486,36.659,156.899
C07938=1041.541,-0.031,419.013,169.488,36.660,156.899
C07939=1041.547,0.219,418.998,169.489,36.661,156.899
C07940=1041.553,0.468,418.983,169.491,36.662,156.899
C07941=1041.559,0.717,418.968,169.493,36.663,156.900
C07942=1041.566,0.967,418.953,169.496,36.663,156.900
C07943=1041.572,1.217,418.938,169.498,36.664,156.900
C07944=1041.578,1.466,418.923,169.500,36.665,156.900
C07945=1041.585,1.716,418.908,169.502,36.666,156.900
C07946=1041.591,1.965,418.894,169.504,36.667,156.901
C07947=1041.597,2.214,418.879,169.506,36.668,156.901
C07948=1041.604,2.464,418.863,169.508,36.668,156.901
C07949=1041.610,2.713,418.848,169.510,36.670,156.901
C07950=1041.616,2.963,418.833,169.512,36.670,156.901
C07951=1041.622,3.212,418.819,169.514,36.671,156.901
C07952=1041.629,3.461,418.804,169.517,36.672,156.902
C07953=1041.635,3.711,418.789,169.518,36.673,156.902
C07954=1041.642,3.960,418.773,169.520,36.674,156.902
C07955=1041.647,4.210,418.758,169.522,36.675,156.902
C07956=1041.654,4.460,418.743,169.524,36.675,156.902
C07957=1041.660,4.709,418.728,169.526,36.677,156.902
C07958=1041.666,4.959,418.713,169.528,36.677,156.902
C07959=1041.673,5.207,418.697,169.530,36.678,156.903
C07960=1041.679,5.457,418.683,169.532,36.679,156.903
C07961=1041.685,5.707,418.668,169.534,36.680,156.903
C07962=1041.692,5.956,418.653,169.537,36.680,156.903
C07963=1041.698,6.205,418.637,169.539,36.682,156.903
C07964=1041.705,6.455,418.622,169.541,36.682,156.903
C07965=1041.711,6.705,418.607,169.542,36.683,156.904
C07966=1041.718,6.954,418.592,169.544,36.684,156.904
C07967=1041.723,7.204,418.576,169.546,36.685,156.904
C07968=1041.730,7.453,418.561,169.548,36.686,156.904
C07969=1041.736,7.703,418.546,169.550,36.687,156.904
C07970=1041.742,7.951,418.531,169.552,36.687,156.904
C07971=1041.749,8.201,418.516,169.554,36.689,156.905
C07972=1041.755,8.451,418.501,169.557,36.689,156.905
C07973=1041.761,8.700,418.486,169.559,36.690,156.905
C07974=1041.768,8.949,418.470,169.561,36.691,156.905
C07975=1041.775,9.199,418.455,169.563,36.692,156.905
C07976=1041.780,9.449,418.440,169.564,36.692,156.905
C07977=1041.787,9.698,418.424,169.566,36.694,156.906
C07978=1041.793,9.948,418.409,169.568,36.694,156.906
C07979=1041.800,10.197,418.393,169.570,36.695,156.906
C07980=1041.806,10.446,418.378,169.572,36.696,156.906
C07981=1041.813,10.696,418.364,169.574,36.697,156.906
C07982=1041.819,10.945,418.348,169.576,36.698,156.906
C07983=1041.826,11.195,418.333,169.579,36.699,156.906
C07984=1041.833,11.444,418.317,169.581,36.699,156.907
C07985=1041.838,11.694,418.302,169.583,36.700,156.907
C07986=1041.845,11.943,418.287,169.585,36.701,156.907
C07987=1041.851,12.192,418.271,169.586,36.702,156.907
C07988=1041.859,12.478,418.253,169.589,36.703,156.907
C07989=1041.866,12.764,418.236,169.591,36.704,156.907
C07990=1041.874,13.049,418.219,169.593,36.705,156.908
C07991=1041.881,13.334,418.201,169.595,36.706,156.908
C07992=1041.887,13.584,418.186,169.598,36.707,156.908
C07993=1041.893,13.833,418.170,169.600,36.708,156.908
C07994=1041.900,14.083,418.155,169.602,36.708,156.908
C07995=1041.906,14.332,418.139,169.604,36.709,156.908
C07996=1041.913,14.581,418.124,169.606,36.710,156.909
C07997=1041.919,14.831,418.108,169.607,36.711,156.909
C07998=1041.925,15.080,418.092,169.609,36.712,156.909
C07999=1041.931,15.330,418.077,169.611,36.713,156.909
C08000=1041.938,15.579,418.061,169.613,36.714,156.909
C08001=1041.944,15.828,418.046,169.616,36.715,156.910
C08002=1041.950,16.078,418.030,169.618,36.716,156.910
C08003=1041.957,16.327,418.014,169.620,36.717,156.910
C08004=1041.962,16.577,417.999,169.621,36.718,156.910
C08005=1041.969,16.826,417.983,169.623,36.719,156.910
C08006=1041.976,17.076,417.968,169.625,36.720,156.910
C08007=1041.982,17.325,417.952,169.627,36.721,156.911
C08008=1041.989,17.575,417.936,169.629,36.721,156.911
C08009=1041.994,17.824,417.920,169.631,36.723,156.911
C08010=1042.001,18.074,417.905,169.634,36.723,156.911
C08011=1042.008,18.323,417.889,169.635,36.725,156.911
C08012=1042.013,18.573,417.874,169.637,36.725,156.911
C08013=1042.020,18.822,417.858,169.639,36.726,156.912
C08014=1042.026,19.071,417.842,169.641,36.727,156.912
C08015=1042.032,19.321,417.827,169.643,36.728,156.912
C08016=1042.039,19.570,417.811,169.645,36.729,156.912
C08017=1042.045,19.819,417.795,169.647,36.730,156.912
C08018=1042.052,20.069,417.779,169.648,36.731,156.913
C08019=1042.058,20.319,417.763,169.651,36.732,156.913
C08020=1042.065,20.568,417.748,169.653,36.733,156.913
C08021=1042.071,20.817,417.731,169.655,36.734,156.913
C08022=1042.077,21.066,417.716,169.657,36.735,156.913
C08023=1042.083,21.316,417.700,169.659,36.736,156.913
C08024=1042.090,21.565,417.684,169.660,36.737,156.914
C08025=1042.096,21.814,417.668,169.662,36.738,156.914
C08026=1042.102,22.064,417.652,169.664,36.738,156.914
C08027=1042.109,22.314,417.636,169.666,36.740,156.914
C08028=1042.115,22.563,417.620,169.669,36.740,156.914
C08029=1042.121,22.813,417.605,169.671,36.742,156.915
C08030=1042.127,23.062,417.588,169.672,36.742,156.915
C08031=1042.134,23.311,417.573,169.674,36.743,156.915
C08032=1042.140,23.560,417.556,169.676,36.744,156.915
C08033=1042.147,23.809,417.541,169.678,36.745,156.915
C08034=1042.153,24.060,417.525,169.680,36.746,156.915
C08035=1042.159,24.309,417.509,169.681,36.747,156.916
C08036=1042.165,24.558,417.493,169.684,36.748,156.916
C08037=1042.171,24.808,417.477,169.686,36.749,156.916
C08038=1042.178,25.057,417.461,169.688,36.750,156.916
C08039=1042.185,25.307,417.444,169.690,36.751,156.916
C08040=1042.191,25.556,417.429,169.692,36.752,156.917
C08041=1042.197,25.805,417.413,169.693,36.753,156.917
C08042=1042.204,26.054,417.397,169.695,36.754,156.917
C08043=1042.210,26.304,417.381,169.697,36.755,156.917
C08044=1042.216,26.554,417.364,169.699,36.756,156.917
C08045=1042.223,26.803,417.349,169.702,36.757,156.917
C08046=1042.229,27.053,417.333,169.704,36.758,156.918
C08047=1042.235,27.302,417.317,169.705,36.759,156.918
C08048=1042.241,27.551,417.301,169.707,36.760,156.918
C08049=1042.248,27.801,417.284,169.709,36.760,156.918
C08050=1042.255,28.050,417.269,169.711,36.762,156.918
C08051=1042.261,28.299,417.252,169.713,36.763,156.919
C08052=1042.268,28.586,417.234,169.715,36.764,156.919
C08053=1042.275,28.872,417.214,169.718,36.765,156.919
C08054=1042.282,29.160,417.196,169.720,36.766,156.919
C08055=1042.290,29.446,417.178,169.722,36.767,156.919
C08056=1042.296,29.695,417.161,169.724,36.769,156.920
C08057=1042.302,29.945,417.145,169.725,36.769,156.920
C08058=1042.308,30.194,417.129,169.727,36.770,156.920
C08059=1042.315,30.444,417.113,169.729,36.772,156.920
C08060=1042.321,30.693,417.096,169.731,36.772,156.920
C08061=1042.327,30.942,417.079,169.734,36.774,156.921
C08062=1042.333,31.191,417.063,169.735,36.774,156.921
C08063=1042.340,31.441,417.047,169.737,36.775,156.921
C08064=1042.346,31.690,417.031,169.739,36.777,156.921
C08065=1042.352,31.940,417.015,169.741,36.777,156.921
C08066=1042.358,32.189,416.998,169.743,36.779,156.922
C08067=1042.365,32.438,416.981,169.744,36.780,156.922
C08068=1042.372,32.688,416.965,169.746,36.780,156.922
C08069=1042.378,32.937,416.949,169.749,36.782,156.922
C08070=1042.384,33.187,416.933,169.751,36.782,156.922
C08071=1042.390,33.436,416.916,169.753,36.784,156.923
C08072=1042.396,33.686,416.900,169.754,36.785,156.923
C08073=1042.402,33.934,416.883,169.756,36.785,156.923
C08074=1042.410,34.184,416.867,169.758,36.787,156.923
C08075=1042.416,34.433,416.851,169.760,36.787,156.923
C08076=1042.422,34.683,416.835,169.762,36.789,156.924
C08077=1042.428,34.933,416.818,169.764,36.790,156.924
C08078=1042.434,35.182,416.801,169.766,36.790,156.924
C08079=1042.441,35.431,416.785,169.768,36.792,156.924
C08080=1042.448,35.681,416.769,169.770,36.792,156.924
C08081=1042.454,35.930,416.752,169.771,36.794,156.924
C08082=1042.460,36.179,416.735,169.773,36.795,156.925
C08083=1042.466,36.429,416.719,169.775,36.795,156.925
C08084=1042.472,36.678,416.703,169.777,36.797,156.925
C08085=1042.479,36.927,416.686,169.779,36.797,156.925
C08086=1042.486,37.177,416.670,169.781,36.799,156.925
C08087=1042.492,37.426,416.653,169.783,36.800,156.926
C08088=1042.498,37.675,416.637,169.785,36.800,156.926
C08089=1042.505,37.925,416.620,169.787,36.802,156.926
C08090=1042.511,38.174,416.603,169.788,36.803,156.926
C08091=1042.517,38.423,416.586,169.790,36.804,156.926
C08092=1042.523,38.673,416.570,169.792,36.805,156.927
C08093=1042.529,38.922,416.554,169.795,36.806,156.927
C08094=1042.536,39.172,416.536,169.797,36.807,156.927
C08095=1042.542,39.421,416.520,169.798,36.808,156.927
C08096=1042.548,39.670,416.504,169.800,36.809,156.927
C08097=1042.554,39.920,416.486,169.802,36.810,156.928
C08098=1042.560,40.169,416.470,169.804,36.811,156.928
C08099=1042.566,40.418,416.453,169.805,36.812,156.928
C08100=1042.573,40.668,416.436,169.807,36.814,156.928
C08101=1042.579,40.917,416.419,169.810,36.814,156.928
C08102=1042.586,41.167,416.402,169.812,36.815,156.929
C08103=1042.592,41.416,416.385,169.813,36.817,156.929
C08104=1042.598,41.665,416.369,169.815,36.818,156.929
C08105=1042.605,41.915,416.353,169.817,36.819,156.929
C08106=1042.611,42.164,416.336,169.819,36.820,156.930
C08107=1042.617,42.414,416.319,169.820,36.821,156.930
C08108=1042.624,42.663,416.302,169.822,36.822,156.930
C08109=1042.630,42.912,416.286,169.825,36.823,156.930
C08110=1042.636,43.161,416.268,169.827,36.824,156.930
C08111=1042.643,43.410,416.251,169.828,36.825,156.930
C08112=1042.649,43.660,416.234,169.830,36.826,156.931
C08113=1042.655,43.909,416.217,169.832,36.827,156.931
C08114=1042.661,44.159,416.201,169.834,36.829,156.931
C08115=1042.667,44.408,416.183,169.835,36.830,156.931
C08116=1042.674,44.695,416.164,169.838,36.831,156.932
C08117=1042.681,44.980,416.144,169.840,36.832,156.932
C08118=1042.688,45.268,416.125,169.842,36.834,156.932
C08119=1042.695,45.554,416.106,169.844,36.835,156.932
C08120=1042.701,45.804,416.088,169.846,36.836,156.933
C08121=1042.708,46.053,416.071,169.848,36.837,156.933
C08122=1042.713,46.302,416.054,169.850,36.838,156.933
C08123=1042.720,46.552,416.037,169.852,36.839,156.933
C08124=1042.726,46.801,416.019,169.854,36.840,156.933
C08125=1042.732,47.051,416.003,169.856,36.842,156.934
C08126=1042.739,47.299,415.986,169.857,36.843,156.934
C08127=1042.745,47.549,415.968,169.859,36.844,156.934
C08128=1042.751,47.798,415.952,169.861,36.845,156.934
C08129=1042.758,48.048,415.934,169.864,36.846,156.935
C08130=1042.763,48.297,415.917,169.865,36.847,156.935
C08131=1042.770,48.546,415.899,169.867,36.849,156.935
C08132=1042.776,48.796,415.883,169.869,36.850,156.935
C08133=1042.781,49.045,415.866,169.870,36.850,156.935
C08134=1042.788,49.294,415.848,169.872,36.852,156.936
C08135=1042.794,49.544,415.832,169.874,36.853,156.936
C08136=1042.800,49.793,415.814,169.877,36.854,156.936
C08137=1042.807,50.042,415.797,169.878,36.855,156.936
C08138=1042.813,50.291,415.780,169.880,36.856,156.937
C08139=1042.819,50.540,415.762,169.882,36.857,156.937
C08140=1042.826,50.791,415.746,169.884,36.859,156.937
C08141=1042.831,51.040,415.728,169.885,36.860,156.937
C08142=1042.838,51.289,415.711,169.887,36.860,156.937
C08143=1042.844,51.538,415.694,169.889,36.862,156.938
C08144=1042.850,51.787,415.676,169.891,36.863,156.938
C08145=1042.857,52.038,415.659,169.893,36.864,156.938
C08146=1042.863,52.286,415.642,169.895,36.865,156.938
C08147=1042.869,52.536,415.624,169.897,36.866,156.938
C08148=1042.875,52.785,415.607,169.898,36.867,156.939
C08149=1042.882,53.034,415.590,169.900,36.869,156.939
C08150=1042.888,53.283,415.572,169.902,36.870,156.939
C08151=1042.894,53.533,415.556,169.905,36.870,156.939
C08152=1042.900,53.782,415.538,169.906,36.872,156.940
C08153=1042.907,54.032,415.521,169.908,36.873,156.940
C08154=1042.914,54.281,415.504,169.910,36.874,156.940
C08155=1042.919,54.530,415.486,169.911,36.875,156.940
C08156=1042.926,54.780,415.469,169.913,36.876,156.940
C08157=1042.932,55.028,415.452,169.915,36.877,156.941
C08158=1042.938,55.278,415.434,169.918,36.878,156.941
C08159=1042.945,55.527,415.416,169.919,36.879,156.941
C08160=1042.951,55.777,415.399,169.921,36.880,156.941
C08161=1042.958,56.026,415.381,169.923,36.882,156.941
C08162=1042.964,56.275,415.365,169.925,36.883,156.942
C08163=1042.970,56.525,415.347,169.926,36.883,156.942
C08164=1042.977,56.774,415.330,169.928,36.885,156.942
C08165=1042.983,57.023,415.313,169.931,36.886,156.942
C08166=1042.989,57.273,415.295,169.933,36.887,156.943
C08167=1042.996,57.522,415.278,169.934,36.888,156.943
C08168=1043.001,57.771,415.260,169.936,36.889,156.943
C08169=1043.008,58.021,415.243,169.938,36.890,156.943
C08170=1043.014,58.270,415.226,169.939,36.892,156.943
C08171=1043.021,58.519,415.208,169.941,36.892,156.944
C08172=1043.027,58.769,415.191,169.943,36.893,156.944
C08173=1043.033,59.018,415.173,169.946,36.895,156.944
C08174=1043.040,59.267,415.156,169.947,36.896,156.944
C08175=1043.047,59.517,415.138,169.949,36.897,156.944
C08176=1043.052,59.765,415.120,169.951,36.898,156.945
C08177=1043.059,60.014,415.103,169.953,36.899,156.945
C08178=1043.065,60.264,415.085,169.954,36.900,156.945
C08179=1043.072,60.514,415.067,169.956,36.901,156.945
C08180=1043.079,60.800,415.047,169.959,36.902,156.945
C08181=1043.087,61.086,415.027,169.961,36.903,156.946
C08182=1043.094,61.372,415.007,169.963,36.905,156.946
C08183=1043.101,61.659,414.987,169.965,36.906,156.946
C08184=1043.108,61.908,414.970,169.967,36.907,156.946
C08185=1043.114,62.157,414.952,169.969,36.908,156.947
C08186=1043.121,62.407,414.935,169.970,36.909,156.947
C08187=1043.127,62.656,414.917,169.973,36.910,156.947
C08188=1043.133,62.905,414.899,169.975,36.911,156.947
C08189=1043.140,63.154,414.882,169.977,36.912,156.947
C08190=1043.146,63.404,414.864,169.978,36.913,156.948
C08191=1043.153,63.653,414.846,169.980,36.914,156.948
C08192=1043.159,63.902,414.829,169.982,36.915,156.948
C08193=1043.166,64.152,414.812,169.984,36.916,156.948
C08194=1043.172,64.401,414.793,169.986,36.918,156.949
C08195=1043.178,64.651,414.775,169.988,36.919,156.949
C08196=1043.184,64.899,414.758,169.990,36.920,156.949
C08197=1043.190,65.149,414.740,169.991,36.921,156.949
C08198=1043.197,65.398,414.721,169.993,36.922,156.949
C08199=1043.202,65.647,414.704,169.995,36.923,156.950
C08200=1043.209,65.897,414.686,169.996,36.924,156.950
C08201=1043.216,66.146,414.668,169.999,36.926,156.950
C08202=1043.222,66.395,414.650,170.001,36.927,156.950
C08203=1043.228,66.644,414.633,170.003,36.928,156.951
C08204=1043.234,66.894,414.615,170.004,36.929,156.951
C08205=1043.241,67.143,414.596,170.006,36.930,156.951
C08206=1043.247,67.392,414.579,170.008,36.931,156.951
C08207=1043.253,67.641,414.561,170.010,36.932,156.951
C08208=1043.259,67.891,414.543,170.012,36.934,156.952
C08209=1043.265,68.140,414.525,170.014,36.935,156.952
C08210=1043.273,68.389,414.507,170.016,36.936,156.952
C08211=1043.278,68.638,414.489,170.017,36.937,156.952
C08212=1043.284,68.888,414.471,170.019,36.938,156.953
C08213=1043.291,69.137,414.453,170.021,36.939,156.953
C08214=1043.298,69.387,414.435,170.023,36.941,156.953
C08215=1043.304,69.636,414.417,170.025,36.942,156.953
C08216=1043.310,69.885,414.399,170.027,36.943,156.953
C08217=1043.316,70.134,414.381,170.029,36.944,156.954
C08218=1043.322,70.384,414.363,170.030,36.945,156.954
C08219=1043.328,70.633,414.345,170.032,36.946,156.954
C08220=1043.334,70.882,414.326,170.034,36.947,156.954
C08221=1043.340,71.131,414.308,170.036,36.949,156.955
C08222=1043.347,71.380,414.290,170.038,36.950,156.955
C08223=1043.353,71.630,414.272,170.040,36.951,156.955
C08224=1043.360,71.879,414.254,170.041,36.952,156.955
C08225=1043.365,72.128,414.236,170.043,36.954,156.956
C08226=1043.372,72.377,414.218,170.045,36.955,156.956
C08227=1043.378,72.627,414.200,170.048,36.956,156.956
C08228=1043.384,72.876,414.181,170.049,36.957,156.956
C08229=1043.390,73.126,414.163,170.051,36.958,156.956
C08230=1043.396,73.374,414.145,170.053,36.959,156.957
C08231=1043.402,73.624,414.127,170.054,36.960,156.957
C08232=1043.409,73.873,414.108,170.056,36.962,156.957
C08233=1043.415,74.123,414.090,170.058,36.963,156.957
C08234=1043.422,74.372,414.072,170.060,36.964,156.958
C08235=1043.429,74.621,414.053,170.062,36.965,156.958
C08236=1043.435,74.871,414.036,170.064,36.967,156.958
C08237=1043.440,75.119,414.017,170.066,36.967,156.958
C08238=1043.447,75.369,413.999,170.067,36.968,156.958
C08239=1043.453,75.618,413.981,170.069,36.970,156.959
C08240=1043.459,75.867,413.962,170.072,36.971,156.959
C08241=1043.466,76.117,413.944,170.073,36.972,156.959
C08242=1043.472,76.366,413.925,170.075,36.973,156.959
C08243=1043.478,76.616,413.908,170.077,36.975,156.960
C08244=1043.485,76.901,413.887,170.079,36.976,156.960
C08245=1043.493,77.187,413.865,170.081,36.977,156.960
C08246=1043.500,77.473,413.845,170.083,36.978,156.960
C08247=1043.507,77.759,413.823,170.086,36.979,156.961
C08248=1043.513,78.009,413.805,170.087,36.981,156.961
C08249=1043.519,78.258,413.786,170.089,36.982,156.961
C08250=1043.526,78.507,413.768,170.091,36.983,156.961
C08251=1043.532,78.756,413.749,170.092,36.984,156.962
C08252=1043.538,79.006,413.731,170.094,36.986,156.962
C08253=1043.544,79.254,413.712,170.097,36.987,156.962
C08254=1043.550,79.504,413.694,170.099,36.988,156.962
C08255=1043.556,79.753,413.675,170.100,36.989,156.963
C08256=1043.563,80.002,413.657,170.102,36.991,156.963
C08257=1043.568,80.252,413.638,170.104,36.992,156.963
C08258=1043.575,80.501,413.619,170.105,36.993,156.963
C08259=1043.581,80.750,413.600,170.108,36.994,156.964
C08260=1043.587,80.999,413.582,170.110,36.996,156.964
C08261=1043.594,81.249,413.564,170.111,36.997,156.964
C08262=1043.599,81.498,413.545,170.113,36.998,156.964
C08263=1043.605,81.747,413.526,170.115,36.999,156.965
C08264=1043.612,81.996,413.508,170.116,37.000,156.965
C08265=1043.618,82.245,413.489,170.119,37.002,156.965
C08266=1043.624,82.494,413.470,170.121,37.003,156.965
C08267=1043.630,82.744,413.451,170.123,37.004,156.966
C08268=1043.636,82.993,413.433,170.124,37.005,156.966
C08269=1043.643,83.242,413.415,170.126,37.007,156.966
C08270=1043.649,83.492,413.396,170.128,37.008,156.966
C08271=1043.655,83.741,413.377,170.130,37.009,156.967
C08272=1043.661,83.990,413.358,170.132,37.010,156.967
C08273=1043.668,84.239,413.339,170.134,37.012,156.967
C08274=1043.674,84.488,413.321,170.135,37.013,156.967
C08275=1043.680,84.738,413.302,170.137,37.014,156.968
C08276=1043.687,84.987,413.283,170.139,37.015,156.968
C08277=1043.693,85.236,413.264,170.141,37.016,156.968
C08278=1043.699,85.485,413.246,170.143,37.017,156.968
C08279=1043.705,85.734,413.227,170.145,37.018,156.968
C08280=1043.712,85.983,413.208,170.147,37.020,156.969
C08281=1043.717,86.233,413.190,170.148,37.021,156.969
C08282=1043.724,86.483,413.171,170.150,37.022,156.969
C08283=1043.730,86.732,413.152,170.152,37.023,156.969
C08284=1043.736,86.981,413.134,170.154,37.025,156.970
C08285=1043.742,87.230,413.115,170.156,37.026,156.970
C08286=1043.749,87.479,413.096,170.158,37.027,156.970
C08287=1043.755,87.729,413.077,170.160,37.028,156.970
C08288=1043.762,87.977,413.058,170.161,37.029,156.971
C08289=1043.767,88.226,413.039,170.163,37.031,156.971
C08290=1043.774,88.476,413.020,170.166,37.032,156.971
C08291=1043.780,88.725,413.001,170.167,37.033,156.971
C08292=1043.787,88.974,412.983,170.169,37.034,156.971
C08293=1043.792,89.223,412.963,170.171,37.035,156.972
C08294=1043.799,89.472,412.945,170.173,37.036,156.972
C08295=1043.805,89.722,412.926,170.174,37.037,156.972
C08296=1043.812,89.971,412.908,170.177,37.039,156.972
C08297=1043.818,90.221,412.888,170.179,37.040,156.973
C08298=1043.824,90.470,412.869,170.181,37.041,156.973
C08299=1043.830,90.719,412.850,170.182,37.042,156.973
C08300=1043.837,90.968,412.831,170.184,37.044,156.973
C08301=1043.843,91.217,412.811,170.186,37.045,156.974
C08302=1043.849,91.466,412.793,170.188,37.046,156.974
C08303=1043.855,91.716,412.774,170.190,37.047,156.974
C08304=1043.861,91.965,412.755,170.192,37.049,156.974
C08305=1043.867,92.214,412.736,170.193,37.050,156.975
C08306=1043.873,92.463,412.716,170.195,37.052,156.975
C08307=1043.879,92.712,412.697,170.197,37.053,156.975
C08308=1043.886,92.999,412.675,170.200,37.054,156.976
C08309=1043.894,93.284,412.653,170.202,37.055,156.976
C08310=1043.901,93.571,412.631,170.204,37.057,156.976
C08311=1043.908,93.856,412.609,170.206,37.058,156.976
C08312=1043.913,94.105,412.590,170.207,37.060,156.977
C08313=1043.920,94.355,412.571,170.210,37.061,156.977
C08314=1043.926,94.604,412.552,170.212,37.062,156.977
C08315=1043.933,94.853,412.533,170.213,37.063,156.977
C08316=1043.939,95.102,412.513,170.215,37.064,156.978
C08317=1043.945,95.351,412.495,170.217,37.066,156.978
C08318=1043.951,95.600,412.475,170.219,37.067,156.978
C08319=1043.957,95.850,412.455,170.221,37.068,156.978
C08320=1043.963,96.099,412.437,170.223,37.069,156.979
C08321=1043.969,96.348,412.417,170.225,37.071,156.979
C08322=1043.976,96.597,412.398,170.226,37.072,156.979
C08323=1043.982,96.847,412.379,170.228,37.073,156.979
C08324=1043.989,97.095,412.359,170.230,37.074,156.980
C08325=1043.994,97.345,412.340,170.233,37.076,156.980
C08326=1044.001,97.594,412.321,170.234,37.077,156.980
C08327=1044.007,97.843,412.301,170.236,37.078,156.980
C08328=1044.014,98.093,412.282,170.238,37.079,156.981
C08329=1044.020,98.341,412.262,170.239,37.080,156.981
C08330=1044.025,98.591,412.243,170.241,37.082,156.981
C08331=1044.032,98.840,412.225,170.244,37.083,156.981
C08332=1044.038,99.089,412.205,170.246,37.084,156.982
C08333=1044.044,99.338,412.186,170.247,37.085,156.982
C08334=1044.051,99.587,412.166,170.249,37.087,156.982
C08335=1044.057,99.836,412.147,170.251,37.088,156.982
C08336=1044.063,100.086,412.128,170.253,37.089,156.983
C08337=1044.070,100.334,412.108,170.255,37.090,156.983
C08338=1044.075,100.584,412.089,170.257,37.091,156.983
C08339=1044.082,100.833,412.069,170.259,37.093,156.983
C08340=1044.088,101.083,412.050,170.260,37.095,156.984
C08341=1044.094,101.332,412.030,170.262,37.096,156.984
C08342=1044.100,101.581,412.011,170.264,37.097,156.984
C08343=1044.106,101.830,411.991,170.267,37.098,156.984
C08344=1044.113,102.079,411.971,170.268,37.099,156.985
C08345=1044.118,102.328,411.951,170.270,37.101,156.985
C08346=1044.124,102.577,411.931,170.272,37.102,156.985
C08347=1044.131,102.826,411.913,170.273,37.104,156.986
C08348=1044.137,103.075,411.893,170.276,37.105,156.986
C08349=1044.142,103.325,411.874,170.278,37.106,156.986
C08350=1044.149,103.574,411.853,170.280,37.107,156.986
C08351=1044.155,103.823,411.833,170.281,37.109,156.987
C08352=1044.161,104.072,411.814,170.283,37.110,156.987
C08353=1044.167,104.321,411.795,170.285,37.111,156.987
C08354=1044.174,104.570,411.774,170.287,37.112,156.987
C08355=1044.180,104.820,411.755,170.289,37.114,156.988
C08356=1044.186,105.069,411.735,170.291,37.115,156.988
C08357=1044.191,105.318,411.716,170.293,37.117,156.988
C08358=1044.199,105.567,411.696,170.294,37.118,156.988
C08359=1044.205,105.816,411.676,170.297,37.119,156.989
C08360=1044.210,106.066,411.657,170.299,37.120,156.989
C08361=1044.216,106.314,411.637,170.301,37.121,156.989
C08362=1044.223,106.564,411.617,170.302,37.123,156.989
C08363=1044.229,106.813,411.597,170.304,37.124,156.990
C08364=1044.235,107.062,411.578,170.306,37.125,156.990
C08365=1044.241,107.311,411.558,170.308,37.126,156.990
C08366=1044.248,107.560,411.538,170.310,37.128,156.990
C08367=1044.254,107.810,411.519,170.312,37.129,156.991
C08368=1044.260,108.058,411.499,170.314,37.131,156.991
C08369=1044.266,108.308,411.478,170.315,37.132,156.991
C08370=1044.272,108.557,411.458,170.317,37.133,156.991
C08371=1044.279,108.806,411.440,170.320,37.134,156.992
C08372=1044.285,109.092,411.417,170.322,37.136,156.992
C08373=1044.293,109.379,411.393,170.324,37.137,156.992
C08374=1044.300,109.664,411.370,170.326,37.139,156.993
C08375=1044.307,109.950,411.347,170.328,37.140,156.993
C08376=1044.313,110.199,411.328,170.331,37.141,156.993
C08377=1044.320,110.448,411.308,170.332,37.142,156.993
C08378=1044.326,110.697,411.289,170.334,37.144,156.994
C08379=1044.332,110.946,411.269,170.336,37.145,156.994
C08380=1044.339,111.195,411.248,170.338,37.147,156.994
C08381=1044.345,111.444,411.228,170.340,37.148,156.994
C08382=1044.350,111.694,411.209,170.342,37.149,156.995
C08383=1044.357,111.943,411.189,170.344,37.150,156.995
C08384=1044.363,112.192,411.169,170.346,37.151,156.995
C08385=1044.369,112.441,411.149,170.347,37.153,156.996
C08386=1044.376,112.690,411.128,170.349,37.155,156.996
C08387=1044.382,112.939,411.108,170.352,37.156,156.996
C08388=1044.388,113.188,411.089,170.354,37.157,156.996
C08389=1044.394,113.438,411.068,170.355,37.158,156.997
C08390=1044.399,113.687,411.048,170.357,37.159,156.997
C08391=1044.405,113.935,411.028,170.359,37.161,156.997
C08392=1044.412,114.185,411.007,170.362,37.162,156.997
C08393=1044.418,114.434,410.987,170.363,37.164,156.998
C08394=1044.423,114.683,410.967,170.365,37.165,156.998
C08395=1044.430,114.932,410.947,170.367,37.167,156.998
C08396=1044.436,115.181,410.927,170.369,37.168,156.999
C08397=1044.442,115.430,410.907,170.371,37.169,156.999
C08398=1044.448,115.680,410.886,170.373,37.170,156.999
C08399=1044.454,115.929,410.866,170.375,37.172,156.999
C08400=1044.460,116.177,410.846,170.376,37.173,157.000
C08401=1044.466,116.427,410.825,170.378,37.175,157.000
C08402=1044.472,116.676,410.805,170.380,37.176,157.000
C08403=1044.478,116.925,410.785,170.383,37.178,157.001
C08404=1044.484,117.174,410.764,170.384,37.179,157.001
C08405=1044.490,117.423,410.743,170.386,37.180,157.001
C08406=1044.496,117.672,410.723,170.388,37.181,157.001
C08407=1044.502,117.921,410.703,170.391,37.183,157.002
C08408=1044.508,118.170,410.683,170.392,37.184,157.002
C08409=1044.514,118.420,410.662,170.394,37.186,157.002
C08410=1044.520,118.669,410.642,170.396,37.187,157.002
C08411=1044.527,118.918,410.622,170.398,37.189,157.003
C08412=1044.532,119.167,410.601,170.399,37.190,157.003
C08413=1044.538,119.416,410.581,170.402,37.191,157.003
C08414=1044.545,119.665,410.560,170.404,37.192,157.004
C08415=1044.550,119.914,410.540,170.406,37.194,157.004
C08416=1044.557,120.164,410.519,170.407,37.195,157.004
C08417=1044.563,120.412,410.499,170.409,37.197,157.004
C08418=1044.570,120.661,410.478,170.412,37.198,157.005
C08419=1044.575,120.911,410.458,170.414,37.200,157.005
C08420=1044.581,121.159,410.438,170.416,37.201,157.005
C08421=1044.587,121.409,410.418,170.417,37.202,157.006
C08422=1044.593,121.657,410.396,170.419,37.203,157.006
C08423=1044.600,121.907,410.376,170.422,37.204,157.006
C08424=1044.606,122.156,410.356,170.424,37.206,157.006
C08425=1044.611,122.406,410.335,170.425,37.208,157.007
C08426=1044.618,122.654,410.314,170.427,37.209,157.007
C08427=1044.624,122.903,410.294,170.429,37.210,157.007
C08428=1044.630,123.152,410.274,170.432,37.212,157.008
C08429=1044.637,123.401,410.253,170.434,37.213,157.008
C08430=1044.643,123.650,410.233,170.435,37.214,157.008
C08431=1044.648,123.900,410.212,170.437,37.215,157.008
C08432=1044.655,124.148,410.191,170.439,37.217,157.009
C08433=1044.661,124.398,410.171,170.442,37.218,157.009
C08434=1044.667,124.647,410.150,170.444,37.220,157.009
C08435=1044.673,124.896,410.129,170.445,37.221,157.009
C08436=1044.680,125.182,410.106,170.447,37.223,157.010
C08437=1044.688,125.468,410.082,170.449,37.224,157.010
C08438=1044.695,125.753,410.058,170.453,37.226,157.010
C08439=1044.702,126.039,410.035,170.455,37.227,157.011
C08440=1044.708,126.288,410.014,170.456,37.228,157.011
C08441=1044.714,126.537,409.994,170.458,37.230,157.011
C08442=1044.720,126.786,409.973,170.460,37.231,157.012
C08443=1044.726,127.036,409.952,170.463,37.232,157.012
C08444=1044.733,127.284,409.931,170.465,37.234,157.012
C08445=1044.739,127.534,409.911,170.466,37.235,157.012
C08446=1044.745,127.782,409.890,170.468,37.237,157.013
C08447=1044.751,128.032,409.869,170.470,37.238,157.013
C08448=1044.757,128.280,409.849,170.473,37.239,157.013
C08449=1044.764,128.530,409.828,170.475,37.240,157.013
C08450=1044.770,128.779,409.807,170.477,37.242,157.014
C08451=1044.776,129.028,409.786,170.478,37.243,157.014
C08452=1044.782,129.277,409.766,170.480,37.245,157.014
C08453=1044.789,129.526,409.745,170.483,37.246,157.015
C08454=1044.794,129.775,409.724,170.485,37.247,157.015
C08455=1044.801,130.024,409.703,170.487,37.248,157.015
C08456=1044.807,130.273,409.683,170.489,37.250,157.015
C08457=1044.814,130.522,409.662,170.490,37.251,157.016
C08458=1044.820,130.772,409.641,170.493,37.252,157.016
C08459=1044.826,131.020,409.620,170.495,37.254,157.016
C08460=1044.833,131.269,409.599,170.497,37.255,157.016
C08461=1044.838,131.519,409.578,170.499,37.257,157.017
C08462=1044.845,131.767,409.557,170.500,37.258,157.017
C08463=1044.851,132.017,409.536,170.502,37.259,157.017
C08464=1044.857,132.266,409.515,170.505,37.261,157.018
C08465=1044.863,132.514,409.494,170.507,37.262,157.018
C08466=1044.869,132.764,409.473,170.509,37.263,157.018
C08467=1044.874,133.013,409.452,170.511,37.265,157.019
C08468=1044.881,133.261,409.431,170.513,37.266,157.019
C08469=1044.887,133.511,409.410,170.515,37.268,157.019
C08470=1044.893,133.760,409.389,170.517,37.269,157.019
C08471=1044.900,134.009,409.368,170.519,37.271,157.020
C08472=1044.906,134.258,409.346,170.521,37.272,157.020
C08473=1044.911,134.507,409.326,170.523,37.274,157.020
C08474=1044.918,134.756,409.304,170.525,37.275,157.021
C08475=1044.924,135.004,409.283,170.527,37.276,157.021
C08476=1044.929,135.254,409.262,170.529,37.278,157.021
C08477=1044.936,135.503,409.241,170.531,37.279,157.021
C08478=1044.942,135.752,409.220,170.534,37.280,157.022
C08479=1044.948,136.001,409.198,170.536,37.282,157.022
C08480=1044.955,136.250,409.177,170.537,37.283,157.022
C08481=1044.961,136.500,409.156,170.539,37.285,157.023
C08482=1044.966,136.748,409.135,170.541,37.286,157.023
C08483=1044.973,136.997,409.113,170.544,37.288,157.023
C08484=1044.979,137.246,409.092,170.546,37.289,157.023
C08485=1044.985,137.495,409.071,170.548,37.291,157.024
C08486=1044.991,137.745,409.050,170.549,37.292,157.024
C08487=1044.997,137.994,409.029,170.551,37.293,157.024
C08488=1045.003,138.242,409.008,170.554,37.295,157.025
C08489=1045.009,138.491,408.986,170.556,37.296,157.025
C08490=1045.016,138.740,408.965,170.558,37.298,157.025
C08491=1045.022,138.990,408.943,170.560,37.299,157.026
C08492=1045.028,139.238,408.922,170.563,37.300,157.026
C08493=1045.034,139.487,408.901,170.564,37.302,157.026
C08494=1045.040,139.737,408.880,170.566,37.303,157.027
C08495=1045.046,139.986,408.858,170.568,37.305,157.027
C08496=1045.052,140.234,408.837,170.570,37.306,157.027
C08497=1045.058,140.484,408.815,170.573,37.308,157.027
C08498=1045.064,140.733,408.794,170.575,37.309,157.028
C08499=1045.070,140.981,408.772,170.577,37.311,157.028
C08500=1045.078,141.267,408.748,170.579,37.312,157.028
C08501=1045.084,141.553,408.723,170.582,37.314,157.029
C08502=1045.091,141.838,408.698,170.584,37.316,157.029
C08503=1045.098,142.123,408.673,170.586,37.317,157.029
C08504=1045.104,142.373,408.651,170.588,37.319,157.030
C08505=1045.111,142.622,408.630,170.590,37.320,157.030
C08506=1045.117,142.871,408.609,170.593,37.322,157.030
C08507=1045.122,143.119,408.588,170.595,37.323,157.031
C08508=1045.129,143.368,408.566,170.596,37.325,157.031
C08509=1045.135,143.618,408.544,170.598,37.326,157.031
C08510=1045.141,143.867,408.523,170.601,37.327,157.032
C08511=1045.147,144.116,408.501,170.603,37.329,157.032
C08512=1045.153,144.365,408.480,170.605,37.330,157.032
C08513=1045.159,144.614,408.458,170.607,37.332,157.033
C08514=1045.165,144.863,408.436,170.609,37.333,157.033
C08515=1045.171,145.112,408.415,170.612,37.335,157.033
C08516=1045.178,145.361,408.392,170.613,37.337,157.033
C08517=1045.183,145.609,408.371,170.615,37.338,157.034
C08518=1045.189,145.858,408.350,170.617,37.340,157.034
C08519=1045.196,146.108,408.328,170.620,37.341,157.034
C08520=1045.202,146.357,408.306,170.622,37.343,157.035
C08521=1045.208,146.606,408.285,170.624,37.344,157.035
C08522=1045.214,146.855,408.262,170.626,37.345,157.035
C08523=1045.220,147.104,408.241,170.628,37.347,157.036
C08524=1045.226,147.352,408.219,170.631,37.348,157.036
C08525=1045.232,147.602,408.198,170.633,37.350,157.036
C08526=1045.238,147.851,408.176,170.634,37.351,157.036
C08527=1045.245,148.099,408.154,170.636,37.353,157.037
C08528=1045.251,148.349,408.132,170.639,37.354,157.037
C08529=1045.257,148.598,408.110,170.641,37.356,157.038
C08530=1045.263,148.846,408.089,170.643,37.357,157.038
C08531=1045.268,149.095,408.066,170.645,37.359,157.038
C08532=1045.275,149.344,408.045,170.647,37.360,157.038
C08533=1045.281,149.594,408.023,170.650,37.362,157.039
C08534=1045.287,149.842,408.001,170.652,37.363,157.039
C08535=1045.293,150.091,407.979,170.654,37.365,157.039
C08536=1045.300,150.341,407.957,170.656,37.367,157.040
C08537=1045.305,150.590,407.934,170.658,37.368,157.040
C08538=1045.311,150.838,407.913,170.660,37.370,157.040
C08539=1045.317,151.087,407.892,170.662,37.371,157.041
C08540=1045.324,151.336,407.869,170.664,37.373,157.041
C08541=1045.329,151.585,407.847,170.667,37.374,157.041
C08542=1045.335,151.834,407.825,170.669,37.376,157.042
C08543=1045.342,152.083,407.803,170.671,37.377,157.042
C08544=1045.348,152.332,407.781,170.673,37.379,157.042
C08545=1045.354,152.581,407.759,170.675,37.380,157.043
C08546=1045.360,152.830,407.737,170.678,37.382,157.043
C08547=1045.366,153.079,407.714,170.680,37.383,157.043
C08548=1045.372,153.328,407.693,170.682,37.385,157.044
C08549=1045.378,153.576,407.671,170.684,37.386,157.044
C08550=1045.384,153.826,407.649,170.687,37.388,157.044
C08551=1045.390,154.074,407.626,170.688,37.390,157.045
C08552=1045.396,154.323,407.605,170.690,37.391,157.045
C08553=1045.403,154.572,407.582,170.692,37.393,157.045
C08554=1045.408,154.822,407.560,170.695,37.394,157.045
C08555=1045.415,155.070,407.538,170.697,37.396,157.046
C08556=1045.421,155.319,407.516,170.699,37.397,157.046
C08557=1045.426,155.568,407.493,170.701,37.398,157.047
C08558=1045.433,155.817,407.471,170.704,37.400,157.047
C08559=1045.439,156.066,407.449,170.706,37.401,157.047
C08560=1045.445,156.315,407.426,170.708,37.403,157.048
C08561=1045.451,156.564,407.404,170.710,37.405,157.048
C08562=1045.457,156.813,407.382,170.713,37.406,157.048
C08563=1045.463,157.062,407.360,170.715,37.408,157.049
C08564=1045.470,157.347,407.334,170.717,37.410,157.049
C08565=1045.477,157.632,407.309,170.719,37.412,157.049
C08566=1045.484,157.918,407.283,170.723,37.414,157.050
C08567=1045.491,158.203,407.258,170.725,37.415,157.050
C08568=1045.497,158.452,407.235,170.727,37.416,157.050
C08569=1045.503,158.701,407.213,170.729,37.418,157.051
C08570=1045.509,158.950,407.190,170.732,37.420,157.051
C08571=1045.515,159.198,407.168,170.734,37.421,157.051
C08572=1045.522,159.448,407.146,170.736,37.423,157.052
C08573=1045.528,159.697,407.123,170.738,37.424,157.052
C08574=1045.534,159.946,407.101,170.741,37.426,157.052
C08575=1045.540,160.195,407.078,170.743,37.428,157.053
C08576=1045.546,160.444,407.056,170.745,37.429,157.053
C08577=1045.552,160.693,407.033,170.747,37.431,157.053
C08578=1045.557,160.942,407.010,170.750,37.433,157.054
C08579=1045.564,161.190,406.988,170.752,37.434,157.054
C08580=1045.570,161.439,406.965,170.753,37.436,157.055
C08581=1045.575,161.688,406.942,170.755,37.438,157.055
C08582=1045.581,161.937,406.920,170.758,37.439,157.055
C08583=1045.587,162.186,406.897,170.760,37.441,157.056
C08584=1045.593,162.435,406.874,170.762,37.443,157.056
C08585=1045.599,162.684,406.851,170.764,37.445,157.056
C08586=1045.604,162.933,406.829,170.767,37.447,157.057
C08587=1045.610,163.182,406.806,170.769,37.448,157.057
C08588=1045.617,163.430,406.783,170.771,37.450,157.057
C08589=1045.622,163.679,406.760,170.773,37.451,157.058
C08590=1045.628,163.928,406.737,170.776,37.453,157.058
C08591=1045.634,164.177,406.714,170.778,37.455,157.058
C08592=1045.640,164.426,406.691,170.780,37.457,157.059
C08593=1045.646,164.674,406.669,170.782,37.458,157.059
C08594=1045.652,164.923,406.646,170.785,37.460,157.060
C08595=1045.657,165.172,406.623,170.787,37.462,157.060
C08596=1045.663,165.421,406.600,170.789,37.463,157.060
C08597=1045.669,165.670,406.577,170.792,37.465,157.061
C08598=1045.675,165.919,406.555,170.794,37.467,157.061
C08599=1045.681,166.167,406.532,170.796,37.468,157.061
C08600=1045.687,166.416,406.509,170.798,37.470,157.062
C08601=1045.693,166.666,406.486,170.801,37.472,157.062
C08602=1045.699,166.915,406.463,170.803,37.473,157.062
C08603=1045.705,167.163,406.440,170.805,37.475,157.063
C08604=1045.711,167.412,406.418,170.807,37.477,157.063
C08605=1045.717,167.661,406.395,170.810,37.478,157.063
C08606=1045.723,167.910,406.372,170.812,37.480,157.064
C08607=1045.728,168.159,406.349,170.814,37.482,157.064
C08608=1045.735,168.408,406.326,170.817,37.484,157.065
C08609=1045.741,168.657,406.302,170.819,37.485,157.065
C08610=1045.747,168.905,406.279,170.821,37.487,157.065
C08611=1045.753,169.154,406.256,170.823,37.488,157.066
C08612=1045.759,169.403,406.233,170.826,37.490,157.066
C08613=1045.764,169.652,406.211,170.828,37.492,157.066
C08614=1045.771,169.901,406.188,170.830,37.494,157.067
C08615=1045.777,170.150,406.165,170.832,37.496,157.067
C08616=1045.783,170.399,406.141,170.835,37.497,157.068
C08617=1045.789,170.648,406.118,170.838,37.499,157.068
C08618=1045.795,170.896,406.095,170.840,37.500,157.068
C08619=1045.800,171.145,406.072,170.842,37.502,157.069
C08620=1045.807,171.394,406.048,170.845,37.504,157.069
C08621=1045.813,171.643,406.026,170.847,37.506,157.069
C08622=1045.819,171.892,406.003,170.849,37.508,157.070
C08623=1045.825,172.141,405.980,170.852,37.509,157.070
C08624=1045.831,172.389,405.956,170.854,37.511,157.071
C08625=1045.837,172.639,405.933,170.856,37.512,157.071
C08626=1045.843,172.887,405.910,170.858,37.514,157.071
C08627=1045.849,173.136,405.887,170.861,37.516,157.072
C08628=1045.857,173.421,405.860,170.864,37.518,157.072
C08629=1045.863,173.706,405.834,170.866,37.520,157.072
C08630=1045.870,173.990,405.807,170.869,37.522,157.073
C08631=1045.877,174.276,405.781,170.872,37.524,157.073
C08632=1045.883,174.525,405.758,170.874,37.525,157.074
C08633=1045.889,174.773,405.734,170.876,37.527,157.074
C08634=1045.895,175.022,405.711,170.879,37.529,157.074
C08635=1045.902,175.271,405.689,170.881,37.531,157.075
C08636=1045.908,175.519,405.665,170.883,37.533,157.075
C08637=1045.914,175.769,405.642,170.885,37.534,157.075
C08638=1045.920,176.017,405.618,170.888,37.536,157.076
C08639=1045.926,176.266,405.595,170.891,37.537,157.076
C08640=1045.932,176.516,405.572,170.893,37.539,157.077
C08641=1045.938,176.764,405.548,170.896,37.541,157.077
C08642=1045.944,177.013,405.525,170.898,37.543,157.077
C08643=1045.951,177.262,405.501,170.900,37.545,157.078
C08644=1045.957,177.510,405.479,170.902,37.546,157.078
C08645=1045.963,177.759,405.455,170.905,37.548,157.078
C08646=1045.970,178.008,405.432,170.907,37.549,157.079
C08647=1045.976,178.257,405.408,170.910,37.551,157.079
C08648=1045.981,178.505,405.385,170.913,37.553,157.080
C08649=1045.988,178.754,405.361,170.915,37.555,157.080
C08650=1045.994,179.003,405.338,170.917,37.556,157.080
C08651=1046.000,179.252,405.314,170.919,37.558,157.081
C08652=1046.006,179.501,405.291,170.922,37.560,157.081
C08653=1046.012,179.749,405.267,170.924,37.562,157.081
C08654=1046.018,179.999,405.244,170.927,37.564,157.082
C08655=1046.025,180.247,405.221,170.930,37.565,157.082
C08656=1046.032,180.496,405.197,170.932,37.566,157.082
C08657=1046.038,180.745,405.174,170.934,37.568,157.083
C08658=1046.044,180.994,405.150,170.936,37.570,157.083
C08659=1046.050,181.243,405.127,170.939,37.572,157.084
C08660=1046.057,181.492,405.103,170.942,37.574,157.084
C08661=1046.063,181.740,405.079,170.944,37.575,157.084
C08662=1046.068,181.989,405.057,170.946,37.577,157.085
C08663=1046.075,182.238,405.032,170.949,37.579,157.085
C08664=1046.081,182.486,405.009,170.951,37.581,157.086
C08665=1046.087,182.736,404.986,170.953,37.583,157.086
C08666=1046.093,182.984,404.962,170.957,37.584,157.086
C08667=1046.100,183.233,404.938,170.959,37.586,157.087
C08668=1046.106,183.482,404.915,170.961,37.587,157.087
C08669=1046.112,183.731,404.891,170.963,37.589,157.087
C08670=1046.118,183.979,404.867,170.966,37.591,157.088
C08671=1046.125,184.228,404.843,170.969,37.593,157.088
C08672=1046.130,184.477,404.820,170.971,37.595,157.089
C08673=1046.137,184.726,404.796,170.974,37.597,157.089
C08674=1046.142,184.975,404.771,170.976,37.599,157.089
C08675=1046.148,185.223,404.748,170.978,37.601,157.090
C08676=1046.154,185.473,404.723,170.981,37.603,157.090
C08677=1046.160,185.721,404.699,170.983,37.604,157.091
C08678=1046.166,185.970,404.675,170.986,37.606,157.091
C08679=1046.172,186.218,404.651,170.989,37.609,157.092
C08680=1046.178,186.468,404.626,170.991,37.610,157.092
C08681=1046.184,186.716,404.603,170.993,37.612,157.092
C08682=1046.189,186.965,404.579,170.995,37.614,157.093
C08683=1046.196,187.214,404.555,170.998,37.616,157.093
C08684=1046.201,187.440,404.533,171.000,37.618,157.094
C08685=1046.206,187.664,404.512,171.002,37.619,157.094
C08686=1046.211,187.890,404.489,171.005,37.621,157.094
C08687=1046.217,188.116,404.467,171.007,37.623,157.095
C08688=1046.223,188.342,404.446,171.009,37.625,157.095
C08689=1046.228,188.567,404.424,171.012,37.626,157.096
C08690=1046.233,188.792,404.402,171.014,37.628,157.096
C08691=1046.239,189.018,404.380,171.016,37.630,157.096
C08692=1046.246,189.349,404.347,171.019,37.632,157.097
C08693=1046.255,189.679,404.316,171.023,37.635,157.097
C08694=1046.263,190.010,404.283,171.026,37.638,157.098
C08695=1046.271,190.342,404.251,171.030,37.641,157.099
C08696=1046.277,190.590,404.227,171.032,37.642,157.099
C08697=1046.283,190.839,404.202,171.034,37.644,157.099
C08698=1046.289,191.087,404.178,171.038,37.646,157.100
C08699=1046.295,191.337,404.154,171.040,37.648,157.100
C08700=1046.301,191.585,404.130,171.042,37.650,157.101
C08701=1046.307,191.834,404.105,171.045,37.652,157.101
C08702=1046.313,192.083,404.081,171.048,37.654,157.102
C08703=1046.319,192.331,404.056,171.050,37.656,157.102
C08704=1046.325,192.580,404.032,171.053,37.658,157.102
C08705=1046.331,192.829,404.008,171.055,37.660,157.103
C08706=1046.337,193.078,403.984,171.058,37.662,157.103
C08707=1046.343,193.326,403.960,171.061,37.664,157.104
C08708=1046.349,193.575,403.935,171.063,37.666,157.104
C08709=1046.356,193.824,403.911,171.065,37.668,157.105
C08710=1046.361,194.073,403.886,171.069,37.670,157.105
C08711=1046.368,194.322,403.862,171.071,37.671,157.105
C08712=1046.374,194.570,403.837,171.073,37.674,157.106
C08713=1046.380,194.818,403.813,171.076,37.676,157.106
C08714=1046.386,195.068,403.789,171.079,37.677,157.107
C08715=1046.392,195.316,403.763,171.081,37.680,157.107
C08716=1046.398,195.565,403.740,171.084,37.682,157.108
C08717=1046.404,195.814,403.715,171.086,37.683,157.108
C08718=1046.411,196.062,403.690,171.089,37.686,157.109
C08719=1046.416,196.311,403.666,171.092,37.687,157.109
C08720=1046.423,196.560,403.642,171.094,37.689,157.109
C08721=1046.429,196.809,403.617,171.097,37.692,157.110
C08722=1046.435,197.057,403.593,171.100,37.693,157.110
C08723=1046.441,197.306,403.568,171.102,37.695,157.111
C08724=1046.447,197.555,403.543,171.105,37.697,157.111
C08725=1046.454,197.804,403.519,171.108,37.699,157.111
C08726=1046.459,198.052,403.494,171.110,37.702,157.112
C08727=1046.466,198.301,403.470,171.112,37.703,157.112
C08728=1046.472,198.549,403.445,171.116,37.705,157.113
C08729=1046.478,198.799,403.420,171.118,37.708,157.113
C08730=1046.485,199.046,403.396,171.120,37.709,157.114
C08731=1046.490,199.296,403.371,171.124,37.711,157.114
C08732=1046.497,199.545,403.347,171.126,37.713,157.115
C08733=1046.503,199.793,403.322,171.128,37.715,157.115
C08734=1046.510,200.042,403.297,171.132,37.718,157.116
C08735=1046.516,200.290,403.273,171.134,37.719,157.116
C08736=1046.522,200.539,403.247,171.136,37.721,157.116
C08737=1046.528,200.788,403.223,171.140,37.723,157.117
C08738=1046.535,201.037,403.198,171.142,37.725,157.117
C08739=1046.540,201.286,403.173,171.144,37.728,157.118
C08740=1046.547,201.533,403.149,171.148,37.729,157.118
C08741=1046.553,201.783,403.124,171.150,37.732,157.119
C08742=1046.559,202.031,403.099,171.152,37.733,157.119
C08743=1046.565,202.280,403.074,171.156,37.736,157.120
C08744=1046.571,202.529,403.049,171.158,37.738,157.120
C08745=1046.577,202.777,403.024,171.161,37.740,157.120
C08746=1046.583,203.026,402.999,171.164,37.742,157.121
C08747=1046.589,203.275,402.973,171.166,37.744,157.121
C08748=1046.595,203.524,402.949,171.169,37.746,157.122
C08749=1046.601,203.773,402.923,171.172,37.749,157.122
C08750=1046.607,204.021,402.898,171.174,37.751,157.123
C08751=1046.614,204.269,402.874,171.177,37.753,157.123
C08752=1046.620,204.518,402.849,171.180,37.755,157.124
C08753=1046.626,204.767,402.824,171.182,37.757,157.124
C08754=1046.632,205.016,402.798,171.186,37.759,157.125
C08755=1046.638,205.264,402.773,171.188,37.761,157.125
C08756=1046.664,206.316,402.667,171.438,37.861,157.149
C08757=1046.671,206.588,402.638,171.440,37.864,157.150
C08758=1046.678,206.858,402.610,171.443,37.867,157.151
C08759=1046.685,207.130,402.582,171.444,37.871,157.151
C08760=1046.692,207.401,402.552,171.447,37.874,157.152
C08761=1046.699,207.650,402.527,171.448,37.877,157.153
C08762=1046.706,207.898,402.500,171.451,37.880,157.153
C08763=1046.711,208.147,402.474,171.453,37.883,157.154
C08764=1046.718,208.395,402.447,171.455,37.886,157.155
C08765=1046.725,208.643,402.421,171.457,37.888,157.155
C08766=1046.731,208.892,402.394,171.459,37.891,157.156
C08767=1046.738,209.140,402.368,171.461,37.894,157.157
C08768=1046.745,209.389,402.342,171.463,37.897,157.157
C08769=1046.751,209.637,402.316,171.465,37.900,157.158
C08770=1046.758,209.886,402.289,171.467,37.903,157.159
C08771=1046.764,210.134,402.263,171.469,37.906,157.159
C08772=1046.770,210.384,402.236,171.472,37.909,157.160
C08773=1046.777,210.632,402.210,171.473,37.912,157.160
C08774=1046.784,210.881,402.184,171.476,37.915,157.161
C08775=1046.790,211.129,402.157,171.477,37.917,157.162
C08776=1046.797,211.378,402.131,171.480,37.920,157.162
C08777=1046.803,211.626,402.104,171.482,37.923,157.163
C08778=1046.810,211.875,402.078,171.484,37.926,157.164
C08779=1046.817,212.123,402.051,171.486,37.929,157.164
C08780=1046.823,212.372,402.024,171.488,37.932,157.165
C08781=1046.829,212.620,401.997,171.491,37.935,157.166
C08782=1046.836,212.869,401.971,171.492,37.938,157.166
C08783=1046.842,213.117,401.944,171.495,37.941,157.167
C08784=1046.849,213.366,401.918,171.497,37.944,157.168
C08785=1046.855,213.614,401.891,171.499,37.947,157.168
C08786=1046.862,213.863,401.865,171.501,37.949,157.169
C08787=1046.867,214.111,401.838,171.503,37.952,157.169
C08788=1046.875,214.359,401.811,171.505,37.955,157.170
C08789=1046.881,214.608,401.784,171.508,37.958,157.171
C08790=1046.887,214.857,401.757,171.509,37.961,157.171
C08791=1046.894,215.105,401.731,171.512,37.964,157.172
C08792=1046.900,215.354,401.704,171.514,37.967,157.173
C08793=1046.907,215.601,401.678,171.516,37.970,157.173
C08794=1046.913,215.850,401.651,171.518,37.973,157.174
C08795=1046.920,216.099,401.624,171.520,37.975,157.174
C08796=1046.926,216.348,401.597,171.522,37.978,157.175
C08797=1046.932,216.597,401.570,171.525,37.981,157.176
C08798=1046.939,216.844,401.544,171.526,37.984,157.176
C08799=1046.946,217.093,401.517,171.529,37.987,157.177
C08800=1046.953,217.342,401.490,171.531,37.990,157.178
C08801=1046.959,217.590,401.463,171.533,37.993,157.178
C08802=1046.965,217.839,401.436,171.535,37.995,157.179
C08803=1046.972,218.087,401.410,171.538,37.998,157.180
C08804=1046.978,218.336,401.383,171.539,38.001,157.180
C08805=1046.985,218.584,401.356,171.542,38.004,157.181
C08806=1046.991,218.832,401.329,171.544,38.007,157.181
C08807=1046.998,219.081,401.303,171.546,38.010,157.182
C08808=1047.005,219.329,401.275,171.548,38.012,157.183
C08809=1047.011,219.578,401.248,171.551,38.015,157.183
C08810=1047.018,219.826,401.221,171.552,38.018,157.184
C08811=1047.025,220.075,401.194,171.555,38.021,157.185
C08812=1047.031,220.323,401.168,171.557,38.024,157.185
C08813=1047.039,220.600,401.138,171.560,38.027,157.186
C08814=1047.045,220.877,401.106,171.563,38.031,157.187
C08815=1047.052,221.153,401.077,171.564,38.034,157.187
C08816=1047.060,221.430,401.046,171.567,38.037,157.188
C08817=1047.065,221.679,401.020,171.569,38.040,157.189
C08818=1047.073,221.927,400.992,171.572,38.043,157.189
C08819=1047.079,222.176,400.965,171.573,38.046,157.190
C08820=1047.085,222.424,400.938,171.576,38.048,157.191
C08821=1047.092,222.673,400.911,171.578,38.051,157.191
C08822=1047.098,222.921,400.883,171.581,38.054,157.192
C08823=1047.104,223.169,400.856,171.582,38.057,157.193
C08824=1047.111,223.418,400.829,171.585,38.060,157.193
C08825=1047.118,223.666,400.802,171.587,38.063,157.194
C08826=1047.124,223.915,400.775,171.589,38.066,157.194
C08827=1047.131,224.163,400.747,171.591,38.069,157.195
C08828=1047.137,224.411,400.720,171.594,38.071,157.196
C08829=1047.144,224.661,400.693,171.596,38.074,157.196
C08830=1047.150,224.908,400.665,171.598,38.077,157.197
C08831=1047.156,225.157,400.638,171.600,38.080,157.198
C08832=1047.163,225.406,400.611,171.603,38.083,157.198
C08833=1047.170,225.653,400.584,171.605,38.086,157.199
C08834=1047.176,225.902,400.557,171.607,38.089,157.200
C08835=1047.183,226.151,400.529,171.610,38.092,157.200
C08836=1047.189,226.399,400.501,171.612,38.094,157.201
C08837=1047.196,226.648,400.474,171.615,38.097,157.201
C08838=1047.202,226.896,400.447,171.616,38.100,157.202
C08839=1047.209,227.144,400.419,171.619,38.103,157.203
C08840=1047.215,227.393,400.392,171.621,38.106,157.203
C08841=1047.222,227.642,400.365,171.624,38.109,157.204
C08842=1047.228,227.889,400.338,171.626,38.111,157.205
C08843=1047.235,228.138,400.310,171.628,38.114,157.205
C08844=1047.242,228.386,400.282,171.630,38.117,157.206
C08845=1047.249,228.635,400.255,171.633,38.120,157.207
C08846=1047.255,228.884,400.228,171.635,38.123,157.207
C08847=1047.262,229.132,400.200,171.637,38.125,157.208
C08848=1047.268,229.380,400.172,171.639,38.128,157.208
C08849=1047.274,229.628,400.145,171.642,38.131,157.209
C08850=1047.281,229.877,400.117,171.644,38.134,157.210
C08851=1047.287,230.125,400.089,171.647,38.137,157.210
C08852=1047.294,230.374,400.061,171.648,38.140,157.211
C08853=1047.299,230.622,400.034,171.651,38.143,157.212
C08854=1047.306,230.871,400.007,171.653,38.145,157.212
C08855=1047.313,231.119,399.979,171.656,38.148,157.213
C08856=1047.319,231.368,399.951,171.658,38.151,157.214
C08857=1047.326,231.616,399.923,171.660,38.154,157.214
C08858=1047.333,231.865,399.896,171.663,38.157,157.215
C08859=1047.338,232.113,399.868,171.665,38.160,157.216
C08860=1047.345,232.361,399.840,171.668,38.163,157.216
C08861=1047.352,232.609,399.812,171.670,38.165,157.217
C08862=1047.358,232.858,399.784,171.673,38.168,157.217
C08863=1047.365,233.106,399.757,171.674,38.171,157.218
C08864=1047.371,233.355,399.728,171.677,38.174,157.219
C08865=1047.377,233.603,399.701,171.679,38.177,157.219
C08866=1047.384,233.851,399.673,171.682,38.180,157.220
C08867=1047.391,234.099,399.645,171.684,38.183,157.221
C08868=1047.397,234.348,399.617,171.687,38.185,157.221
C08869=1047.402,234.559,399.593,171.688,38.188,157.222
C08870=1047.408,234.769,399.569,171.691,38.190,157.223
C08871=1047.413,234.980,399.546,171.692,38.193,157.223
C08872=1047.419,235.191,399.522,171.695,38.195,157.224
C08873=1047.424,235.402,399.498,171.696,38.197,157.224
C08874=1047.429,235.611,399.475,171.699,38.200,157.225
C08875=1047.435,235.822,399.451,171.701,38.202,157.225
C08876=1047.441,236.033,399.427,171.702,38.204,157.226
C08877=1047.447,236.281,399.399,171.705,38.207,157.226
C08878=1047.453,236.530,399.371,171.708,38.210,157.227
C08879=1047.460,236.778,399.343,171.710,38.213,157.228
C08880=1047.467,237.027,399.316,171.713,38.216,157.228
C08881=1047.473,237.275,399.287,171.714,38.219,157.229
C08882=1047.480,237.523,399.259,171.717,38.222,157.230
C08883=1047.486,237.772,399.231,171.719,38.224,157.230
C08884=1047.493,238.020,399.203,171.722,38.227,157.231
C08885=1047.502,238.365,399.164,171.726,38.231,157.232
C08886=1047.511,238.709,399.125,171.728,38.235,157.233
C08887=1047.520,239.054,399.085,171.732,38.239,157.234
C08888=1047.529,239.399,399.047,171.736,38.243,157.235
C08889=1047.535,239.647,399.019,171.738,38.246,157.235
C08890=1047.542,239.895,398.990,171.741,38.249,157.236
C08891=1047.548,240.144,398.962,171.742,38.251,157.236
C08892=1047.555,240.392,398.933,171.745,38.254,157.237
C08893=1047.561,240.640,398.905,171.747,38.257,157.238
C08894=1047.568,240.889,398.878,171.750,38.260,157.238
C08895=1047.574,241.137,398.849,171.753,38.263,157.239
C08896=1047.581,241.385,398.821,171.755,38.266,157.240
C08897=1047.587,241.633,398.792,171.758,38.268,157.240
C08898=1047.594,241.882,398.764,171.760,38.271,157.241
C08899=1047.600,242.130,398.735,171.763,38.274,157.242
C08900=1047.607,242.378,398.707,171.765,38.277,157.242
C08901=1047.613,242.626,398.678,171.768,38.279,157.243
C08902=1047.619,242.875,398.650,171.770,38.282,157.244
C08903=1047.626,243.123,398.622,171.773,38.285,157.244
C08904=1047.632,243.372,398.593,171.776,38.288,157.245
C08905=1047.639,243.620,398.565,171.778,38.291,157.246
C08906=1047.645,243.869,398.536,171.781,38.294,157.246
C08907=1047.652,244.117,398.507,171.782,38.296,157.247
C08908=1047.659,244.365,398.479,171.785,38.299,157.247
C08909=1047.665,244.614,398.450,171.787,38.302,157.248
C08910=1047.671,244.862,398.422,171.790,38.305,157.249
C08911=1047.678,245.110,398.393,171.792,38.308,157.249
C08912=1047.684,245.358,398.365,171.795,38.311,157.250
C08913=1047.691,245.606,398.336,171.797,38.314,157.251
C08914=1047.697,245.854,398.307,171.800,38.317,157.252
C08915=1047.703,246.103,398.279,171.803,38.320,157.252
C08916=1047.709,246.351,398.250,171.805,38.323,157.253
C08917=1047.715,246.599,398.221,171.808,38.325,157.254
C08918=1047.722,246.847,398.192,171.810,38.328,157.254
C08919=1047.728,247.096,398.164,171.813,38.331,157.255
C08920=1047.735,247.344,398.135,171.815,38.334,157.256
C08921=1047.741,247.593,398.105,171.818,38.337,157.256
C08922=1047.748,247.841,398.076,171.821,38.340,157.257
C08923=1047.754,248.089,398.047,171.823,38.343,157.258
C08924=1047.760,248.338,398.019,171.826,38.345,157.258
C08925=1047.767,248.601,397.988,171.828,38.349,157.259
C08926=1047.774,248.864,397.958,171.831,38.352,157.260
C08927=1047.780,249.127,397.927,171.833,38.355,157.260
C08928=1047.787,249.391,397.897,171.837,38.358,157.261
C08929=1047.794,249.639,397.868,171.840,38.361,157.262
C08930=1047.800,249.888,397.839,171.842,38.363,157.262
C08931=1047.806,250.136,397.810,171.845,38.366,157.263
C08932=1047.813,250.385,397.780,171.847,38.369,157.264
C08933=1047.819,250.633,397.751,171.850,38.372,157.264
C08934=1047.825,250.881,397.722,171.852,38.375,157.265
C08935=1047.832,251.129,397.694,171.855,38.378,157.266
C08936=1047.839,251.377,397.665,171.858,38.381,157.266
C08937=1047.845,251.626,397.635,171.860,38.384,157.267
C08938=1047.852,251.874,397.606,171.863,38.386,157.268
C08939=1047.858,252.122,397.577,171.865,38.389,157.268
C08940=1047.864,252.370,397.548,171.868,38.392,157.269
C08941=1047.870,252.618,397.519,171.870,38.395,157.270
C08942=1047.877,252.867,397.490,171.873,38.398,157.270
C08943=1047.884,253.115,397.461,171.876,38.401,157.271
C08944=1047.890,253.363,397.432,171.878,38.404,157.272
C08945=1047.897,253.611,397.403,171.881,38.407,157.272
C08946=1047.904,253.860,397.374,171.883,38.409,157.273
C08947=1047.910,254.108,397.345,171.887,38.412,157.274
C08948=1047.916,254.356,397.315,171.889,38.415,157.274
C08949=1047.923,254.604,397.286,171.892,38.418,157.275
C08950=1047.930,254.852,397.257,171.895,38.421,157.276
C08951=1047.936,255.101,397.227,171.897,38.423,157.276
C08952=1047.942,255.349,397.198,171.900,38.426,157.277
C08953=1047.948,255.597,397.169,171.902,38.429,157.278
C08954=1047.955,255.845,397.139,171.905,38.432,157.278
C08955=1047.962,256.093,397.110,171.907,38.435,157.279
C08956=1047.968,256.341,397.081,171.910,38.438,157.280
C08957=1047.975,256.590,397.052,171.914,38.441,157.280
C08958=1047.981,256.838,397.023,171.916,38.443,157.281
C08959=1047.988,257.086,396.994,171.919,38.446,157.282
C08960=1047.995,257.334,396.964,171.921,38.449,157.282
C08961=1048.001,257.582,396.935,171.924,38.452,157.283
C08962=1048.008,257.830,396.905,171.926,38.455,157.284
C08963=1048.015,258.079,396.876,171.929,38.457,157.284
C08964=1048.021,258.327,396.847,171.933,38.460,157.285
C08965=1048.028,258.576,396.818,171.935,38.463,157.286
C08966=1048.035,258.823,396.788,171.938,38.466,157.286
C08967=1048.041,259.071,396.759,171.940,38.469,157.287
C08968=1048.048,259.320,396.729,171.943,38.471,157.288
C08969=1048.054,259.568,396.700,171.945,38.474,157.288
C08970=1048.061,259.817,396.670,171.949,38.477,157.289
C08971=1048.068,260.064,396.640,171.952,38.480,157.290
C08972=1048.074,260.312,396.611,171.954,38.483,157.290
C08973=1048.081,260.561,396.582,171.957,38.486,157.291
C08974=1048.087,260.809,396.552,171.959,38.489,157.292
C08975=1048.094,261.057,396.523,171.963,38.491,157.292
C08976=1048.101,261.305,396.493,171.965,38.494,157.293
C08977=1048.108,261.554,396.464,171.968,38.497,157.294
C08978=1048.114,261.801,396.434,171.971,38.499,157.294
C08979=1048.121,262.050,396.404,171.973,38.502,157.295
C08980=1048.127,262.298,396.375,171.977,38.505,157.296
C08981=1048.134,262.560,396.344,171.979,38.508,157.296
C08982=1048.141,262.821,396.313,171.982,38.511,157.297
C08983=1048.148,263.083,396.282,171.986,38.514,157.298
C08984=1048.155,263.345,396.249,171.988,38.517,157.298
C08985=1048.162,263.594,396.220,171.991,38.520,157.299
C08986=1048.168,263.842,396.189,171.993,38.523,157.300
C08987=1048.175,264.090,396.159,171.996,38.526,157.300
C08988=1048.181,264.338,396.130,172.000,38.529,157.301
C08989=1048.188,264.587,396.100,172.002,38.532,157.302
C08990=1048.194,264.834,396.070,172.005,38.534,157.303
C08991=1048.201,265.082,396.040,172.007,38.537,157.303
C08992=1048.207,265.331,396.010,172.011,38.541,157.304
C08993=1048.213,265.578,395.980,172.014,38.544,157.305
C08994=1048.220,265.826,395.950,172.016,38.546,157.305
C08995=1048.226,266.074,395.920,172.019,38.549,157.306
C08996=1048.233,266.323,395.890,172.021,38.552,157.307
C08997=1048.240,266.571,395.861,172.025,38.555,157.307
C08998=1048.246,266.819,395.830,172.028,38.558,157.308
C08999=1048.253,267.067,395.800,172.030,38.561,157.309
C09000=1048.260,267.315,395.770,172.033,38.564,157.309
C09001=1048.266,267.564,395.740,172.036,38.566,157.310
C09002=1048.272,267.812,395.710,172.039,38.569,157.311
C09003=1048.279,268.060,395.680,172.042,38.572,157.312
C09004=1048.285,268.308,395.650,172.045,38.575,157.312
C09005=1048.292,268.556,395.619,172.048,38.578,157.313
C09006=1048.298,268.804,395.589,172.050,38.581,157.314
C09007=1048.306,269.052,395.559,172.053,38.584,157.314
C09008=1048.311,269.300,395.529,172.057,38.586,157.315
C09009=1048.319,269.548,395.499,172.059,38.590,157.316
C09010=1048.324,269.796,395.468,172.062,38.593,157.316
C09011=1048.332,270.044,395.438,172.064,38.596,157.317
C09012=1048.338,270.292,395.408,172.068,38.598,157.318
C09013=1048.344,270.540,395.377,172.071,38.601,157.319
C09014=1048.351,270.788,395.347,172.073,38.604,157.319
C09015=1048.357,271.036,395.317,172.077,38.607,157.320
C09016=1048.364,271.284,395.287,172.079,38.610,157.321
C09017=1048.370,271.533,395.256,172.082,38.613,157.321
C09018=1048.377,271.781,395.226,172.086,38.616,157.322
C09019=1048.383,272.029,395.195,172.088,38.619,157.323
C09020=1048.390,272.277,395.165,172.091,38.622,157.323
C09021=1048.397,272.524,395.134,172.094,38.625,157.324
C09022=1048.403,272.773,395.104,172.097,38.628,157.325
C09023=1048.410,273.020,395.074,172.100,38.630,157.326
C09024=1048.416,273.269,395.043,172.102,38.633,157.326
C09025=1048.422,273.518,395.012,172.106,38.637,157.327
C09026=1048.429,273.764,394.982,172.109,38.640,157.328
C09027=1048.436,274.013,394.951,172.111,38.642,157.328
C09028=1048.442,274.261,394.920,172.115,38.645,157.329
C09029=1048.449,274.509,394.891,172.118,38.648,157.330
C09030=1048.455,274.757,394.859,172.120,38.652,157.331
C09031=1048.462,275.005,394.829,172.124,38.654,157.331
C09032=1048.468,275.253,394.798,172.126,38.657,157.332
C09033=1048.475,275.501,394.767,172.129,38.660,157.333
C09034=1048.481,275.749,394.737,172.133,38.663,157.333
C09035=1048.487,275.997,394.706,172.135,38.666,157.334
C09036=1048.494,276.245,394.675,172.139,38.669,157.335
C09037=1048.501,276.512,394.643,172.142,38.672,157.336
C09038=1048.508,276.778,394.609,172.145,38.675,157.336
C09039=1048.515,277.043,394.576,172.148,38.679,157.337
C09040=1048.522,277.310,394.543,172.152,38.682,157.338
C09041=1048.529,277.558,394.513,172.154,38.685,157.339
C09042=1048.536,277.806,394.481,172.158,38.688,157.339
C09043=1048.542,278.054,394.451,172.161,38.691,157.340
C09044=1048.548,278.302,394.420,172.163,38.694,157.341
C09045=1048.555,278.550,394.389,172.167,38.696,157.342
C09046=1048.562,278.798,394.359,172.170,38.699,157.342
C09047=1048.569,279.046,394.327,172.173,38.703,157.343
C09048=1048.575,279.293,394.296,172.176,38.706,157.344
C09049=1048.581,279.542,394.265,172.178,38.708,157.344
C09050=1048.588,279.790,394.234,172.182,38.712,157.345
C09051=1048.594,280.038,394.203,172.185,38.715,157.346
C09052=1048.601,280.286,394.172,172.188,38.717,157.347
C09053=1048.607,280.533,394.141,172.191,38.720,157.347
C09054=1048.614,280.782,394.110,172.194,38.724,157.348
C09055=1048.620,281.030,394.079,172.197,38.727,157.349
C09056=1048.627,281.278,394.047,172.200,38.729,157.350
C09057=1048.633,281.526,394.017,172.204,38.733,157.350
C09058=1048.640,281.774,393.985,172.206,38.736,157.351
C09059=1048.646,282.021,393.954,172.210,38.738,157.352
C09060=1048.653,282.269,393.923,172.213,38.742,157.353
C09061=1048.660,282.518,393.892,172.215,38.745,157.353
C09062=1048.666,282.765,393.861,172.219,38.748,157.354
C09063=1048.672,283.013,393.829,172.222,38.751,157.355
C09064=1048.679,283.261,393.798,172.225,38.754,157.355
C09065=1048.686,283.509,393.766,172.228,38.757,157.356
C09066=1048.692,283.757,393.736,172.232,38.760,157.357
C09067=1048.699,284.005,393.704,172.234,38.763,157.358
C09068=1048.706,284.253,393.673,172.238,38.766,157.359
C09069=1048.712,284.501,393.641,172.241,38.769,157.359
C09070=1048.719,284.748,393.610,172.244,38.772,157.360
C09071=1048.725,284.996,393.579,172.247,38.775,157.361
C09072=1048.732,285.244,393.548,172.251,38.778,157.361
C09073=1048.739,285.492,393.516,172.253,38.781,157.362
C09074=1048.745,285.740,393.485,172.257,38.784,157.363
C09075=1048.751,285.989,393.453,172.260,38.787,157.364
C09076=1048.758,286.237,393.422,172.263,38.790,157.364
C09077=1048.765,286.484,393.390,172.266,38.793,157.365
C09078=1048.771,286.732,393.359,172.270,38.796,157.366
C09079=1048.778,286.980,393.328,172.272,38.800,157.367
C09080=1048.785,287.228,393.296,172.276,38.802,157.367
C09081=1048.792,287.476,393.265,172.279,38.805,157.368
C09082=1048.798,287.724,393.233,172.282,38.809,157.369
C09083=1048.805,287.971,393.201,172.285,38.811,157.370
C09084=1048.811,288.219,393.169,172.289,38.815,157.370
C09085=1048.818,288.467,393.138,172.291,38.818,157.371
C09086=1048.825,288.715,393.106,172.295,38.821,157.372
C09087=1048.831,288.963,393.075,172.298,38.824,157.373
C09088=1048.837,289.211,393.043,172.302,38.827,157.374
C09089=1048.844,289.459,393.011,172.304,38.830,157.374
C09090=1048.851,289.707,392.979,172.308,38.833,157.375
C09091=1048.858,289.954,392.948,172.312,38.836,157.376
C09092=1048.864,290.203,392.916,172.314,38.840,157.377
C09093=1048.872,290.480,392.880,172.318,38.843,157.377
C09094=1048.878,290.758,392.845,172.322,38.846,157.378
C09095=1048.886,291.035,392.809,172.326,38.850,157.379
C09096=1048.894,291.313,392.774,172.329,38.853,157.380
C09097=1048.900,291.561,392.741,172.332,38.856,157.381
C09098=1048.907,291.808,392.710,172.336,38.859,157.382
C09099=1048.913,292.057,392.677,172.338,38.863,157.382
C09100=1048.920,292.305,392.645,172.342,38.865,157.383
C09101=1048.927,292.553,392.614,172.346,38.869,157.384
C09102=1048.933,292.801,392.582,172.349,38.872,157.385
C09103=1048.940,293.048,392.550,172.352,38.875,157.385
C09104=1048.947,293.296,392.518,172.355,38.878,157.386
C09105=1048.953,293.543,392.485,172.359,38.881,157.387
